LIN {X 0,Y 469.267,Z 468.198,A -85,B 0,C 180,E1 -7456.775,E2 -7456.775} C_VEL
LIN {X 0,Y 468.626,Z 477.541,A -85,B 0,C 180,E1 -7458.1,E2 -7458.1} C_VEL
LIN {X 0,Y 468.005,Z 486.29,A -85,B 0,C 180,E1 -7459.618,E2 -7459.618} C_VEL
LIN {X 0,Y 467.579,Z 492.456,A -85,B 0,C 180,E1 -7460.919,E2 -7460.919} C_VEL
LIN {X 0,Y 467.288,Z 497.539,A -85,B 0,C 180,E1 -7462.22,E2 -7462.22} C_VEL
LIN {X 0,Y 467.051,Z 502.915,A -85,B 0,C 180,E1 -7463.953,E2 -7463.953} C_VEL
LIN {X 0,Y 466.841,Z 506.814,A -85,B 0,C 180,E1 -7465.683,E2 -7465.683} C_VEL
LIN {X 0,Y 466.764,Z 509.357,A -85,B 0,C 180,E1 -7467.411,E2 -7467.411} C_VEL
LIN {X 0,Y 466.622,Z 510.634,A -85,B 0,C 180,E1 -7469.137,E2 -7469.137} C_VEL
LIN {X 0,Y 466.622,Z 510.669,A -85,B 0,C 180,E1 -7470.863,E2 -7470.863} C_VEL
LIN {X 0,Y 466.762,Z 509.467,A -85,B 0,C 180,E1 -7472.589,E2 -7472.589} C_VEL
LIN {X 0,Y 466.825,Z 506.997,A -85,B 0,C 180,E1 -7474.317,E2 -7474.317} C_VEL
LIN {X 0,Y 467.046,Z 503.165,A -85,B 0,C 180,E1 -7476.046,E2 -7476.046} C_VEL
LIN {X 0,Y 467.237,Z 497.87,A -85,B 0,C 180,E1 -7477.78,E2 -7477.78} C_VEL
LIN {X 0,Y 467.649,Z 490.923,A -85,B 0,C 180,E1 -7479.515,E2 -7479.515} C_VEL
LIN {X 0,Y 468.194,Z 483.257,A -85,B 0,C 180,E1 -7481.033,E2 -7481.033} C_VEL
LIN {X 0,Y 468.792,Z 475.255,A -85,B 0,C 180,E1 -7482.335,E2 -7482.335} C_VEL
LIN {X 0,Y 469.426,Z 465.627,A -85,B 0,C 180,E1 -7483.638,E2 -7483.638} C_VEL
LIN {X 0,Y 470.223,Z 454.915,A -85,B 0,C 180,E1 -7484.829,E2 -7484.829} C_VEL
LIN {X 0,Y 471,Z 443.033,A -85,B 0,C 180,E1 -7485.913,E2 -7485.913} C_VEL
LIN {X 0,Y 471.72,Z 431.29,A -85,B 0,C 180,E1 -7486.777,E2 -7486.777} C_VEL
LIN {X 0,Y 472.372,Z 418.989,A -85,B 0,C 180,E1 -7487.5,E2 -7487.5} C_VEL
LIN {X 0,Y 472.878,Z 404.897,A -85,B 0,C 180,E1 -7488.135,E2 -7488.135} C_VEL
LIN {X 0,Y 473.318,Z 391.368,A -85,B 0,C 180,E1 -7488.56,E2 -7488.56} C_VEL
LIN {X 0,Y 473.564,Z 375.614,A -85,B 0,C 180,E1 -7488.859,E2 -7488.859} C_VEL
LIN {X 0,Y 474.304,Z 263.513,A -85,B 0,C 180,E1 -7490.488,E2 -7490.488} C_VEL
LIN {X 0,Y 470.511,Z 244.594,A -85,B 0,C 180,E1 -7490.98,E2 -7490.98} C_VEL
LIN {X 0,Y 470.717,Z 239.725,A -85,B 0,C 180,E1 -7491.686,E2 -7491.686} C_VEL
LIN {X 0,Y 472.048,Z 216.347,A -85,B 0,C 180,E1 -7495.342,E2 -7495.342} C_VEL
LIN {X 0,Y 471.922,Z 212.053,A -85,B 0,C 180,E1 -7496.045,E2 -7496.045} C_VEL
LIN {X 0,Y 468.466,Z 197.446,A -85,B 0,C 180,E1 -7498.689,E2 -7498.689} C_VEL
LIN {X 0,Y 467.573,Z 193.923,A -85,B 0,C 180,E1 -7499.4,E2 -7499.4} C_VEL
LIN {X 0,Y 467.582,Z 193.852,A -85,B 0,C 180,E1 -7502.758,E2 -7502.758} C_VEL
LIN {X 0,Y 467.554,Z 193.869,A -85,B 0,C 180,E1 -7505.889,E2 -7505.889} C_VEL
LIN {X 0,Y 467.58,Z 193.863,A -85,B 0,C 180,E1 -7509.144,E2 -7509.144} C_VEL
LIN {X 0,Y 467.583,Z 193.858,A -85,B 0,C 180,E1 -7512.566,E2 -7512.566} C_VEL
LIN {X 0,Y 467.567,Z 193.867,A -85,B 0,C 180,E1 -7515.052,E2 -7515.052} C_VEL
LIN {X 0,Y 467.585,Z 193.867,A -85,B 0,C 180,E1 -7517.439,E2 -7517.439} C_VEL
LIN {X 0,Y 467.556,Z 193.86,A -85,B 0,C 180,E1 -7520.852,E2 -7520.852} C_VEL
LIN {X 0,Y 467.558,Z 193.862,A -85,B 0,C 180,E1 -7524.26,E2 -7524.26} C_VEL
LIN {X 0,Y 467.577,Z 193.868,A -85,B 0,C 180,E1 -7527.32,E2 -7527.32} C_VEL
LIN {X 0,Y 467.573,Z 193.857,A -85,B 0,C 180,E1 -7530.665,E2 -7530.665} C_VEL
LIN {X 0,Y 467.611,Z 193.86,A -85,B 0,C 180,E1 -7533.199,E2 -7533.199} C_VEL
LIN {X 0,Y 467.586,Z 193.861,A -85,B 0,C 180,E1 -7536.468,E2 -7536.468} C_VEL
LIN {X 0,Y 467.616,Z 193.854,A -85,B 0,C 180,E1 -7539.777,E2 -7539.777} C_VEL
LIN {X 0,Y 467.603,Z 193.864,A -85,B 0,C 180,E1 -7542.506,E2 -7542.506} C_VEL
LIN {X 0,Y 467.601,Z 193.863,A -85,B 0,C 180,E1 -7545.196,E2 -7545.196} C_VEL
LIN {X 0,Y 467.649,Z 193.851,A -85,B 0,C 180,E1 -7547.854,E2 -7547.854} C_VEL
LIN {X 0,Y 467.675,Z 193.849,A -85,B 0,C 180,E1 -7551.357,E2 -7551.357} C_VEL
LIN {X 0,Y 467.736,Z 193.843,A -85,B 0,C 180,E1 -7553.962,E2 -7553.962} C_VEL
LIN {X 0,Y 467.853,Z 193.826,A -85,B 0,C 180,E1 -7557.417,E2 -7557.417} C_VEL
LIN {X 0,Y 467.875,Z 193.829,A -85,B 0,C 180,E1 -7560,E2 -7560} C_VEL
LIN {X 0,Y 467.853,Z 193.834,A -85,B 0,C 180,E1 -7562.583,E2 -7562.583} C_VEL
LIN {X 0,Y 467.736,Z 193.843,A -85,B 0,C 180,E1 -7566.037,E2 -7566.037} C_VEL
LIN {X 0,Y 467.674,Z 193.851,A -85,B 0,C 180,E1 -7568.643,E2 -7568.643} C_VEL
LIN {X 0,Y 467.648,Z 193.86,A -85,B 0,C 180,E1 -7572.145,E2 -7572.145} C_VEL
LIN {X 0,Y 467.631,Z 193.859,A -85,B 0,C 180,E1 -7575.695,E2 -7575.695} C_VEL
LIN {X 0,Y 467.61,Z 193.858,A -85,B 0,C 180,E1 -7578.765,E2 -7578.765} C_VEL
LIN {X 0,Y 467.573,Z 193.863,A -85,B 0,C 180,E1 -7581.268,E2 -7581.268} C_VEL
LIN {X 0,Y 467.566,Z 193.867,A -85,B 0,C 180,E1 -7583.943,E2 -7583.943} C_VEL
LIN {X 0,Y 467.612,Z 193.845,A -85,B 0,C 180,E1 -7586.8,E2 -7586.8} C_VEL
LIN {X 0,Y 467.546,Z 193.873,A -85,B 0,C 180,E1 -7589.739,E2 -7589.739} C_VEL
LIN {X 0,Y 467.577,Z 193.851,A -85,B 0,C 180,E1 -7592.759,E2 -7592.759} C_VEL
LIN {X 0,Y 467.55,Z 193.867,A -85,B 0,C 180,E1 -7595.89,E2 -7595.89} C_VEL
LIN {X 0,Y 467.576,Z 193.864,A -85,B 0,C 180,E1 -7599.145,E2 -7599.145} C_VEL
LIN {X 0,Y 467.581,Z 193.859,A -85,B 0,C 180,E1 -7602.567,E2 -7602.567} C_VEL
LIN {X 0,Y 467.56,Z 193.867,A -85,B 0,C 180,E1 -7605.053,E2 -7605.053} C_VEL
LIN {X 0,Y 467.584,Z 193.867,A -85,B 0,C 180,E1 -7607.441,E2 -7607.441} C_VEL
LIN {X 0,Y 467.554,Z 193.848,A -85,B 0,C 180,E1 -7610.853,E2 -7610.853} C_VEL
LIN {X 0,Y 467.555,Z 193.855,A -85,B 0,C 180,E1 -7614.262,E2 -7614.262} C_VEL
LIN {X 0,Y 467.569,Z 193.861,A -85,B 0,C 180,E1 -7617.323,E2 -7617.323} C_VEL
LIN {X 0,Y 467.574,Z 194.014,A -85,B 0,C 180,E1 -7619.018,E2 -7619.018} C_VEL
LIN {X 0,Y 470.497,Z 204.521,A -85,B 0,C 180,E1 -7620.713,E2 -7620.713} C_VEL
LIN {X 0,Y 473.464,Z 217.047,A -85,B 0,C 180,E1 -7622.604,E2 -7622.604} C_VEL
LIN {X 0,Y 471.777,Z 243.748,A -85,B 0,C 180,E1 -7626.051,E2 -7626.051} C_VEL
LIN {X 0,Y 471.739,Z 245.311,A -85,B 0,C 180,E1 -7626.211,E2 -7626.211} C_VEL
LIN {X 0,Y 475.092,Z 265.679,A -85,B 0,C 180,E1 -7626.729,E2 -7626.729} C_VEL
LIN {X 0,Y 473.209,Z 408.687,A -85,B 0,C 180,E1 -7629.062,E2 -7629.062} C_VEL
LIN {X 0,Y 472.673,Z 424.604,A -85,B 0,C 180,E1 -7629.491,E2 -7629.491} C_VEL
LIN {X 0,Y 472.053,Z 439.866,A -85,B 0,C 180,E1 -7630.089,E2 -7630.089} C_VEL
LIN {X 0,Y 471.299,Z 454.544,A -85,B 0,C 180,E1 -7630.849,E2 -7630.849} C_VEL
LIN {X 0,Y 470.534,Z 467.938,A -85,B 0,C 180,E1 -7631.721,E2 -7631.721} C_VEL
LIN {X 0,Y 469.794,Z 481.582,A -85,B 0,C 180,E1 -7632.816,E2 -7632.816} C_VEL
LIN {X 0,Y 469.075,Z 493.997,A -85,B 0,C 180,E1 -7634.02,E2 -7634.02} C_VEL
LIN {X 0,Y 468.418,Z 504.464,A -85,B 0,C 180,E1 -7635.223,E2 -7635.223} C_VEL
LIN {X 0,Y 467.834,Z 515.629,A -85,B 0,C 180,E1 -7636.757,E2 -7636.757} C_VEL
LIN {X 0,Y 467.425,Z 524.894,A -85,B 0,C 180,E1 -7638.289,E2 -7638.289} C_VEL
LIN {X 0,Y 467.087,Z 532.575,A -85,B 0,C 180,E1 -7639.817,E2 -7639.817} C_VEL
LIN {X 0,Y 466.875,Z 538.894,A -85,B 0,C 180,E1 -7641.343,E2 -7641.343} C_VEL
LIN {X 0,Y 466.758,Z 544.686,A -85,B 0,C 180,E1 -7643.082,E2 -7643.082} C_VEL
LIN {X 0,Y 466.717,Z 549.068,A -85,B 0,C 180,E1 -7644.817,E2 -7644.817} C_VEL
LIN {X 0,Y 466.706,Z 552.142,A -85,B 0,C 180,E1 -7646.547,E2 -7646.547} C_VEL
LIN {X 0,Y 466.658,Z 553.973,A -85,B 0,C 180,E1 -7648.274,E2 -7648.274} C_VEL
LIN {X 0,Y 466.597,Z 554.595,A -85,B 0,C 180,E1 -7650,E2 -7650} C_VEL
LIN {X 0,Y 466.658,Z 553.97,A -85,B 0,C 180,E1 -7651.726,E2 -7651.726} C_VEL
LIN {X 0,Y 466.706,Z 552.136,A -85,B 0,C 180,E1 -7653.454,E2 -7653.454} C_VEL
LIN {X 0,Y 466.722,Z 549.065,A -85,B 0,C 180,E1 -7655.184,E2 -7655.184} C_VEL
LIN {X 0,Y 466.821,Z 544.69,A -85,B 0,C 180,E1 -7656.918,E2 -7656.918} C_VEL
LIN {X 0,Y 466.875,Z 538.89,A -85,B 0,C 180,E1 -7658.658,E2 -7658.658} C_VEL
LIN {X 0,Y 467.179,Z 531.526,A -85,B 0,C 180,E1 -7660.4,E2 -7660.4} C_VEL
LIN {X 0,Y 467.477,Z 523.63,A -85,B 0,C 180,E1 -7661.93,E2 -7661.93} C_VEL
LIN {X 0,Y 467.919,Z 514.123,A -85,B 0,C 180,E1 -7663.462,E2 -7663.462} C_VEL
LIN {X 0,Y 468.413,Z 504.449,A -85,B 0,C 180,E1 -7664.778,E2 -7664.778} C_VEL
LIN {X 0,Y 469.096,Z 492.954,A -85,B 0,C 180,E1 -7666.091,E2 -7666.091} C_VEL
LIN {X 0,Y 469.869,Z 480.323,A -85,B 0,C 180,E1 -7667.294,E2 -7667.294} C_VEL
LIN {X 0,Y 470.543,Z 467.908,A -85,B 0,C 180,E1 -7668.28,E2 -7668.28} C_VEL
LIN {X 0,Y 471.313,Z 454.501,A -85,B 0,C 180,E1 -7669.151,E2 -7669.151} C_VEL
LIN {X 0,Y 472.067,Z 439.828,A -85,B 0,C 180,E1 -7669.911,E2 -7669.911} C_VEL
LIN {X 0,Y 472.701,Z 424.193,A -85,B 0,C 180,E1 -7670.521,E2 -7670.521} C_VEL
LIN {X 0,Y 473.161,Z 408.552,A -85,B 0,C 180,E1 -7670.941,E2 -7670.941} C_VEL
LIN {X 0,Y 475.017,Z 270.123,A -85,B 0,C 180,E1 -7673.198,E2 -7673.198} C_VEL
LIN {X 0,Y 474.917,Z 264.066,A -85,B 0,C 180,E1 -7673.304,E2 -7673.304} C_VEL
LIN {X 0,Y 471.704,Z 245.037,A -85,B 0,C 180,E1 -7673.801,E2 -7673.801} C_VEL
LIN {X 0,Y 473.005,Z 224.215,A -85,B 0,C 180,E1 -7676.471,E2 -7676.471} C_VEL
LIN {X 0,Y 473.439,Z 217.06,A -85,B 0,C 180,E1 -7677.399,E2 -7677.399} C_VEL
LIN {X 0,Y 470.952,Z 206.283,A -85,B 0,C 180,E1 -7679.012,E2 -7679.012} C_VEL
LIN {X 0,Y 467.576,Z 193.975,A -85,B 0,C 180,E1 -7680.983,E2 -7680.983} C_VEL
LIN {X 0,Y 467.575,Z 193.857,A -85,B 0,C 180,E1 -7684.24,E2 -7684.24} C_VEL
LIN {X 0,Y 467.546,Z 193.873,A -85,B 0,C 180,E1 -7687.186,E2 -7687.186} C_VEL
LIN {X 0,Y 467.572,Z 193.842,A -85,B 0,C 180,E1 -7690.265,E2 -7690.265} C_VEL
LIN {X 0,Y 467.585,Z 193.867,A -85,B 0,C 180,E1 -7692.567,E2 -7692.567} C_VEL
LIN {X 0,Y 467.564,Z 193.867,A -85,B 0,C 180,E1 -7695.052,E2 -7695.052} C_VEL
LIN {X 0,Y 467.587,Z 193.858,A -85,B 0,C 180,E1 -7697.44,E2 -7697.44} C_VEL
LIN {X 0,Y 467.58,Z 193.864,A -85,B 0,C 180,E1 -7700.855,E2 -7700.855} C_VEL
LIN {X 0,Y 467.557,Z 193.869,A -85,B 0,C 180,E1 -7704.261,E2 -7704.261} C_VEL
LIN {X 0,Y 467.579,Z 193.851,A -85,B 0,C 180,E1 -7707.321,E2 -7707.321} C_VEL
LIN {X 0,Y 467.566,Z 193.867,A -85,B 0,C 180,E1 -7710.668,E2 -7710.668} C_VEL
LIN {X 0,Y 467.61,Z 193.844,A -85,B 0,C 180,E1 -7713.199,E2 -7713.199} C_VEL
LIN {X 0,Y 467.588,Z 193.866,A -85,B 0,C 180,E1 -7716.469,E2 -7716.469} C_VEL
LIN {X 0,Y 467.62,Z 193.859,A -85,B 0,C 180,E1 -7719.777,E2 -7719.777} C_VEL
LIN {X 0,Y 467.605,Z 193.861,A -85,B 0,C 180,E1 -7722.507,E2 -7722.507} C_VEL
LIN {X 0,Y 467.603,Z 193.859,A -85,B 0,C 180,E1 -7725.197,E2 -7725.197} C_VEL
LIN {X 0,Y 467.653,Z 193.859,A -85,B 0,C 180,E1 -7727.855,E2 -7727.855} C_VEL
LIN {X 0,Y 467.678,Z 193.85,A -85,B 0,C 180,E1 -7731.357,E2 -7731.357} C_VEL
LIN {X 0,Y 467.74,Z 193.843,A -85,B 0,C 180,E1 -7733.963,E2 -7733.963} C_VEL
LIN {X 0,Y 467.856,Z 193.833,A -85,B 0,C 180,E1 -7737.417,E2 -7737.417} C_VEL
LIN {X 0,Y 467.879,Z 193.829,A -85,B 0,C 180,E1 -7740,E2 -7740} C_VEL
LIN {X 0,Y 467.857,Z 193.825,A -85,B 0,C 180,E1 -7742.583,E2 -7742.583} C_VEL
LIN {X 0,Y 467.741,Z 193.843,A -85,B 0,C 180,E1 -7746.038,E2 -7746.038} C_VEL
LIN {X 0,Y 467.679,Z 193.849,A -85,B 0,C 180,E1 -7748.643,E2 -7748.643} C_VEL
LIN {X 0,Y 467.653,Z 193.85,A -85,B 0,C 180,E1 -7752.146,E2 -7752.146} C_VEL
LIN {X 0,Y 467.637,Z 193.854,A -85,B 0,C 180,E1 -7755.695,E2 -7755.695} C_VEL
LIN {X 0,Y 467.615,Z 193.861,A -85,B 0,C 180,E1 -7758.765,E2 -7758.765} C_VEL
LIN {X 0,Y 467.578,Z 193.869,A -85,B 0,C 180,E1 -7761.268,E2 -7761.268} C_VEL
LIN {X 0,Y 467.57,Z 193.862,A -85,B 0,C 180,E1 -7763.944,E2 -7763.944} C_VEL
LIN {X 0,Y 467.615,Z 193.861,A -85,B 0,C 180,E1 -7766.801,E2 -7766.801} C_VEL
LIN {X 0,Y 467.552,Z 193.86,A -85,B 0,C 180,E1 -7769.738,E2 -7769.738} C_VEL
LIN {X 0,Y 467.582,Z 193.867,A -85,B 0,C 180,E1 -7772.759,E2 -7772.759} C_VEL
LIN {X 0,Y 467.556,Z 193.861,A -85,B 0,C 180,E1 -7775.89,E2 -7775.89} C_VEL
LIN {X 0,Y 467.559,Z 193.859,A -85,B 0,C 180,E1 -7779.147,E2 -7779.147} C_VEL
LIN {X 0,Y 467.586,Z 193.868,A -85,B 0,C 180,E1 -7782.567,E2 -7782.567} C_VEL
LIN {X 0,Y 467.571,Z 193.867,A -85,B 0,C 180,E1 -7785.053,E2 -7785.053} C_VEL
LIN {X 0,Y 467.589,Z 193.858,A -85,B 0,C 180,E1 -7787.44,E2 -7787.44} C_VEL
LIN {X 0,Y 467.582,Z 193.862,A -85,B 0,C 180,E1 -7790.856,E2 -7790.856} C_VEL
LIN {X 0,Y 467.562,Z 193.869,A -85,B 0,C 180,E1 -7794.261,E2 -7794.261} C_VEL
LIN {X 0,Y 467.583,Z 193.851,A -85,B 0,C 180,E1 -7797.321,E2 -7797.321} C_VEL
LIN {X 0,Y 467.586,Z 193.972,A -85,B 0,C 180,E1 -7800.732,E2 -7800.732} C_VEL
LIN {X 0,Y 470.786,Z 207.019,A -85,B 0,C 180,E1 -7803.155,E2 -7803.155} C_VEL
LIN {X 0,Y 472.11,Z 212.897,A -85,B 0,C 180,E1 -7804.201,E2 -7804.201} C_VEL
LIN {X 0,Y 471.337,Z 227.381,A -85,B 0,C 180,E1 -7806.493,E2 -7806.493} C_VEL
LIN {X 0,Y 470.478,Z 244.431,A -85,B 0,C 180,E1 -7809.102,E2 -7809.102} C_VEL
LIN {X 0,Y 474.392,Z 264.64,A -85,B 0,C 180,E1 -7809.626,E2 -7809.626} C_VEL
LIN {X 0,Y 474.417,Z 267.518,A -85,B 0,C 180,E1 -7809.67,E2 -7809.67} C_VEL
LIN {X 0,Y 473.774,Z 273.373,A -85,B 0,C 180,E1 -7809.728,E2 -7809.728} C_VEL
LIN {X 0,Y 468.182,Z 292.425,A -85,B 0,C 180,E1 -7809.744,E2 -7809.744} C_VEL
LIN {X 0,Y 467.551,Z 298.281,A -85,B 0,C 180,E1 -7809.802,E2 -7809.802} C_VEL
LIN {X 0,Y 466.805,Z 384.962,A -85,B 0,C 180,E1 -7811.085,E2 -7811.085} C_VEL
LIN {X 0,Y 466.403,Z 399.475,A -85,B 0,C 180,E1 -7811.467,E2 -7811.467} C_VEL
LIN {X 0,Y 465.951,Z 413.371,A -85,B 0,C 180,E1 -7812.023,E2 -7812.023} C_VEL
LIN {X 0,Y 465.404,Z 425.207,A -85,B 0,C 180,E1 -7812.648,E2 -7812.648} C_VEL
LIN {X 0,Y 464.569,Z 438.207,A -85,B 0,C 180,E1 -7813.522,E2 -7813.522} C_VEL
LIN {X 0,Y 463.756,Z 449.946,A -85,B 0,C 180,E1 -7814.508,E2 -7814.508} C_VEL
LIN {X 0,Y 463.052,Z 459.693,A -85,B 0,C 180,E1 -7815.497,E2 -7815.497} C_VEL
LIN {X 0,Y 462.234,Z 470.42,A -85,B 0,C 180,E1 -7816.817,E2 -7816.817} C_VEL
LIN {X 0,Y 461.554,Z 479.282,A -85,B 0,C 180,E1 -7818.137,E2 -7818.137} C_VEL
LIN {X 0,Y 460.921,Z 487.753,A -85,B 0,C 180,E1 -7819.679,E2 -7819.679} C_VEL
LIN {X 0,Y 460.444,Z 494.611,A -85,B 0,C 180,E1 -7821.22,E2 -7821.22} C_VEL
LIN {X 0,Y 460.07,Z 500.781,A -85,B 0,C 180,E1 -7822.98,E2 -7822.98} C_VEL
LIN {X 0,Y 459.882,Z 504.367,A -85,B 0,C 180,E1 -7824.299,E2 -7824.299} C_VEL
LIN {X 0,Y 459.752,Z 507.157,A -85,B 0,C 180,E1 -7825.616,E2 -7825.616} C_VEL
LIN {X 0,Y 459.683,Z 509.694,A -85,B 0,C 180,E1 -7827.371,E2 -7827.371} C_VEL
LIN {X 0,Y 459.556,Z 510.966,A -85,B 0,C 180,E1 -7829.123,E2 -7829.123} C_VEL
LIN {X 0,Y 459.556,Z 511.001,A -85,B 0,C 180,E1 -7830.876,E2 -7830.876} C_VEL
LIN {X 0,Y 459.68,Z 509.802,A -85,B 0,C 180,E1 -7832.629,E2 -7832.629} C_VEL
LIN {X 0,Y 459.736,Z 507.339,A -85,B 0,C 180,E1 -7834.383,E2 -7834.383} C_VEL
LIN {X 0,Y 460.001,Z 503.513,A -85,B 0,C 180,E1 -7836.139,E2 -7836.139} C_VEL
LIN {X 0,Y 460.209,Z 498.228,A -85,B 0,C 180,E1 -7837.899,E2 -7837.899} C_VEL
LIN {X 0,Y 460.535,Z 493.23,A -85,B 0,C 180,E1 -7839.22,E2 -7839.22} C_VEL
LIN {X 0,Y 461.08,Z 486.029,A -85,B 0,C 180,E1 -7840.761,E2 -7840.761} C_VEL
LIN {X 0,Y 461.627,Z 478.513,A -85,B 0,C 180,E1 -7842.083,E2 -7842.083} C_VEL
LIN {X 0,Y 462.328,Z 468.945,A -85,B 0,C 180,E1 -7843.479,E2 -7843.479} C_VEL
LIN {X 0,Y 463.096,Z 458.514,A -85,B 0,C 180,E1 -7844.726,E2 -7844.726} C_VEL
LIN {X 0,Y 463.91,Z 447.333,A -85,B 0,C 180,E1 -7845.824,E2 -7845.824} C_VEL
LIN {X 0,Y 464.779,Z 434.949,A -85,B 0,C 180,E1 -7846.809,E2 -7846.809} C_VEL
LIN {X 0,Y 465.402,Z 422.958,A -85,B 0,C 180,E1 -7847.578,E2 -7847.578} C_VEL
LIN {X 0,Y 466.095,Z 409.337,A -85,B 0,C 180,E1 -7848.248,E2 -7848.248} C_VEL
LIN {X 0,Y 466.529,Z 395.19,A -85,B 0,C 180,E1 -7848.755,E2 -7848.755} C_VEL
LIN {X 0,Y 466.852,Z 380.668,A -85,B 0,C 180,E1 -7849.083,E2 -7849.083} C_VEL
LIN {X 0,Y 467.834,Z 265.856,A -85,B 0,C 180,E1 -7850.771,E2 -7850.771} C_VEL
LIN {X 0,Y 463.8,Z 245.038,A -85,B 0,C 180,E1 -7851.306,E2 -7851.306} C_VEL
LIN {X 0,Y 463.686,Z 243.548,A -85,B 0,C 180,E1 -7851.447,E2 -7851.447} C_VEL
LIN {X 0,Y 464.914,Z 222.567,A -85,B 0,C 180,E1 -7854.762,E2 -7854.762} C_VEL
LIN {X 0,Y 465.323,Z 215.002,A -85,B 0,C 180,E1 -7855.976,E2 -7855.976} C_VEL
LIN {X 0,Y 461.978,Z 200.465,A -85,B 0,C 180,E1 -7858.632,E2 -7858.632} C_VEL
LIN {X 0,Y 460.532,Z 194.804,A -85,B 0,C 180,E1 -7859.758,E2 -7859.758} C_VEL
LIN {X 0,Y 460.529,Z 194.728,A -85,B 0,C 180,E1 -7862.929,E2 -7862.929} C_VEL
LIN {X 0,Y 460.498,Z 194.746,A -85,B 0,C 180,E1 -7866.014,E2 -7866.014} C_VEL
LIN {X 0,Y 460.542,Z 194.74,A -85,B 0,C 180,E1 -7868.897,E2 -7868.897} C_VEL
LIN {X 0,Y 460.52,Z 194.739,A -85,B 0,C 180,E1 -7872.181,E2 -7872.181} C_VEL
LIN {X 0,Y 460.513,Z 194.742,A -85,B 0,C 180,E1 -7875.411,E2 -7875.411} C_VEL
LIN {X 0,Y 460.528,Z 194.743,A -85,B 0,C 180,E1 -7878.397,E2 -7878.397} C_VEL
LIN {X 0,Y 460.514,Z 194.741,A -85,B 0,C 180,E1 -7881.266,E2 -7881.266} C_VEL
LIN {X 0,Y 460.509,Z 194.741,A -85,B 0,C 180,E1 -7884.554,E2 -7884.554} C_VEL
LIN {X 0,Y 460.527,Z 194.744,A -85,B 0,C 180,E1 -7887.715,E2 -7887.715} C_VEL
LIN {X 0,Y 460.542,Z 194.731,A -85,B 0,C 180,E1 -7890.769,E2 -7890.769} C_VEL
LIN {X 0,Y 460.557,Z 194.738,A -85,B 0,C 180,E1 -7893.734,E2 -7893.734} C_VEL
LIN {X 0,Y 460.54,Z 194.74,A -85,B 0,C 180,E1 -7896.623,E2 -7896.623} C_VEL
LIN {X 0,Y 460.544,Z 194.737,A -85,B 0,C 180,E1 -7899.452,E2 -7899.452} C_VEL
LIN {X 0,Y 460.553,Z 194.739,A -85,B 0,C 180,E1 -7902.23,E2 -7902.23} C_VEL
LIN {X 0,Y 460.559,Z 194.742,A -85,B 0,C 180,E1 -7904.964,E2 -7904.964} C_VEL
LIN {X 0,Y 460.602,Z 194.729,A -85,B 0,C 180,E1 -7907.665,E2 -7907.665} C_VEL
LIN {X 0,Y 460.622,Z 194.729,A -85,B 0,C 180,E1 -7911.224,E2 -7911.224} C_VEL
LIN {X 0,Y 460.703,Z 194.719,A -85,B 0,C 180,E1 -7913.87,E2 -7913.87} C_VEL
LIN {X 0,Y 460.818,Z 194.702,A -85,B 0,C 180,E1 -7917.377,E2 -7917.377} C_VEL
LIN {X 0,Y 460.845,Z 194.704,A -85,B 0,C 180,E1 -7920,E2 -7920} C_VEL
LIN {X 0,Y 460.818,Z 194.71,A -85,B 0,C 180,E1 -7922.622,E2 -7922.622} C_VEL
LIN {X 0,Y 460.703,Z 194.719,A -85,B 0,C 180,E1 -7926.13,E2 -7926.13} C_VEL
LIN {X 0,Y 460.621,Z 194.728,A -85,B 0,C 180,E1 -7928.776,E2 -7928.776} C_VEL
LIN {X 0,Y 460.606,Z 194.733,A -85,B 0,C 180,E1 -7932.445,E2 -7932.445} C_VEL
LIN {X 0,Y 460.592,Z 194.74,A -85,B 0,C 180,E1 -7935.998,E2 -7935.998} C_VEL
LIN {X 0,Y 460.563,Z 194.736,A -85,B 0,C 180,E1 -7938.902,E2 -7938.902} C_VEL
LIN {X 0,Y 460.508,Z 194.744,A -85,B 0,C 180,E1 -7941.486,E2 -7941.486} C_VEL
LIN {X 0,Y 460.536,Z 194.739,A -85,B 0,C 180,E1 -7944.332,E2 -7944.332} C_VEL
LIN {X 0,Y 460.573,Z 194.723,A -85,B 0,C 180,E1 -7947.244,E2 -7947.244} C_VEL
LIN {X 0,Y 460.503,Z 194.745,A -85,B 0,C 180,E1 -7950.24,E2 -7950.24} C_VEL
LIN {X 0,Y 460.523,Z 194.734,A -85,B 0,C 180,E1 -7953.325,E2 -7953.325} C_VEL
LIN {X 0,Y 460.472,Z 194.746,A -85,B 0,C 180,E1 -7956.53,E2 -7956.53} C_VEL
LIN {X 0,Y 460.552,Z 194.742,A -85,B 0,C 180,E1 -7959.86,E2 -7959.86} C_VEL
LIN {X 0,Y 460.506,Z 194.742,A -85,B 0,C 180,E1 -7962.901,E2 -7962.901} C_VEL
LIN {X 0,Y 460.503,Z 194.743,A -85,B 0,C 180,E1 -7965.831,E2 -7965.831} C_VEL
LIN {X 0,Y 460.525,Z 194.728,A -85,B 0,C 180,E1 -7968.989,E2 -7968.989} C_VEL
LIN {X 0,Y 460.513,Z 194.73,A -85,B 0,C 180,E1 -7971.267,E2 -7971.267} C_VEL
LIN {X 0,Y 460.504,Z 194.73,A -85,B 0,C 180,E1 -7974.555,E2 -7974.555} C_VEL
LIN {X 0,Y 460.514,Z 194.719,A -85,B 0,C 180,E1 -7977.715,E2 -7977.715} C_VEL
LIN {X 0,Y 460.577,Z 194.958,A -85,B 0,C 180,E1 -7978.662,E2 -7978.662} C_VEL
LIN {X 0,Y 464.137,Z 208.021,A -85,B 0,C 180,E1 -7980.777,E2 -7980.777} C_VEL
LIN {X 0,Y 466.622,Z 218.341,A -85,B 0,C 180,E1 -7982.366,E2 -7982.366} C_VEL
LIN {X 0,Y 465.289,Z 240.561,A -85,B 0,C 180,E1 -7985.294,E2 -7985.294} C_VEL
LIN {X 0,Y 464.98,Z 245.065,A -85,B 0,C 180,E1 -7985.857,E2 -7985.857} C_VEL
LIN {X 0,Y 468.54,Z 267.054,A -85,B 0,C 180,E1 -7986.431,E2 -7986.431} C_VEL
LIN {X 0,Y 466.521,Z 408.803,A -85,B 0,C 180,E1 -7988.776,E2 -7988.776} C_VEL
LIN {X 0,Y 465.944,Z 424.716,A -85,B 0,C 180,E1 -7989.215,E2 -7989.215} C_VEL
LIN {X 0,Y 465.359,Z 439.202,A -85,B 0,C 180,E1 -7989.79,E2 -7989.79} C_VEL
LIN {X 0,Y 464.533,Z 453.968,A -85,B 0,C 180,E1 -7990.559,E2 -7990.559} C_VEL
LIN {X 0,Y 463.725,Z 467.409,A -85,B 0,C 180,E1 -7991.443,E2 -7991.443} C_VEL
LIN {X 0,Y 462.909,Z 481.098,A -85,B 0,C 180,E1 -7992.552,E2 -7992.552} C_VEL
LIN {X 0,Y 462.183,Z 492.772,A -85,B 0,C 180,E1 -7993.69,E2 -7993.69} C_VEL
LIN {X 0,Y 461.456,Z 504.023,A -85,B 0,C 180,E1 -7994.995,E2 -7994.995} C_VEL
LIN {X 0,Y 460.832,Z 515.218,A -85,B 0,C 180,E1 -7996.552,E2 -7996.552} C_VEL
LIN {X 0,Y 460.351,Z 524.661,A -85,B 0,C 180,E1 -7998.137,E2 -7998.137} C_VEL
LIN {X 0,Y 460.06,Z 532.193,A -85,B 0,C 180,E1 -7999.66,E2 -7999.66} C_VEL
LIN {X 0,Y 459.81,Z 538.525,A -85,B 0,C 180,E1 -8001.209,E2 -8001.209} C_VEL
LIN {X 0,Y 459.69,Z 544.329,A -85,B 0,C 180,E1 -8002.975,E2 -8002.975} C_VEL
LIN {X 0,Y 459.622,Z 548.721,A -85,B 0,C 180,E1 -8004.736,E2 -8004.736} C_VEL
LIN {X 0,Y 459.601,Z 551.802,A -85,B 0,C 180,E1 -8006.494,E2 -8006.494} C_VEL
LIN {X 0,Y 459.567,Z 553.639,A -85,B 0,C 180,E1 -8008.248,E2 -8008.248} C_VEL
LIN {X 0,Y 459.528,Z 554.263,A -85,B 0,C 180,E1 -8010,E2 -8010} C_VEL
LIN {X 0,Y 459.567,Z 553.636,A -85,B 0,C 180,E1 -8011.753,E2 -8011.753} C_VEL
LIN {X 0,Y 459.601,Z 551.796,A -85,B 0,C 180,E1 -8013.507,E2 -8013.507} C_VEL
LIN {X 0,Y 459.633,Z 548.717,A -85,B 0,C 180,E1 -8015.264,E2 -8015.264} C_VEL
LIN {X 0,Y 459.728,Z 544.331,A -85,B 0,C 180,E1 -8017.025,E2 -8017.025} C_VEL
LIN {X 0,Y 459.811,Z 538.519,A -85,B 0,C 180,E1 -8018.792,E2 -8018.792} C_VEL
LIN {X 0,Y 460.102,Z 531.138,A -85,B 0,C 180,E1 -8020.562,E2 -8020.562} C_VEL
LIN {X 0,Y 460.446,Z 522.769,A -85,B 0,C 180,E1 -8022.196,E2 -8022.196} C_VEL
LIN {X 0,Y 460.935,Z 513.702,A -85,B 0,C 180,E1 -8023.67,E2 -8023.67} C_VEL
LIN {X 0,Y 461.447,Z 504.004,A -85,B 0,C 180,E1 -8025.006,E2 -8025.006} C_VEL
LIN {X 0,Y 462.118,Z 492.743,A -85,B 0,C 180,E1 -8026.313,E2 -8026.313} C_VEL
LIN {X 0,Y 463.007,Z 479.814,A -85,B 0,C 180,E1 -8027.559,E2 -8027.559} C_VEL
LIN {X 0,Y 463.744,Z 467.371,A -85,B 0,C 180,E1 -8028.557,E2 -8028.557} C_VEL
LIN {X 0,Y 464.544,Z 453.916,A -85,B 0,C 180,E1 -8029.441,E2 -8029.441} C_VEL
LIN {X 0,Y 465.309,Z 439.145,A -85,B 0,C 180,E1 -8030.213,E2 -8030.213} C_VEL
LIN {X 0,Y 466.003,Z 423.834,A -85,B 0,C 180,E1 -8030.812,E2 -8030.812} C_VEL
LIN {X 0,Y 466.473,Z 408.654,A -85,B 0,C 180,E1 -8031.227,E2 -8031.227} C_VEL
LIN {X 0,Y 468.214,Z 286.116,A -85,B 0,C 180,E1 -8033.258,E2 -8033.258} C_VEL
LIN {X 0,Y 468.341,Z 265.157,A -85,B 0,C 180,E1 -8033.608,E2 -8033.608} C_VEL
LIN {X 0,Y 464.97,Z 245.006,A -85,B 0,C 180,E1 -8034.145,E2 -8034.145} C_VEL
LIN {X 0,Y 466.625,Z 220.822,A -85,B 0,C 180,E1 -8037.3,E2 -8037.3} C_VEL
LIN {X 0,Y 466.355,Z 216.897,A -85,B 0,C 180,E1 -8037.851,E2 -8037.851} C_VEL
LIN {X 0,Y 462.711,Z 202.567,A -85,B 0,C 180,E1 -8040.081,E2 -8040.081} C_VEL
LIN {X 0,Y 460.536,Z 194.836,A -85,B 0,C 180,E1 -8041.37,E2 -8041.37} C_VEL
LIN {X 0,Y 460.521,Z 194.731,A -85,B 0,C 180,E1 -8044.504,E2 -8044.504} C_VEL
LIN {X 0,Y 460.499,Z 194.747,A -85,B 0,C 180,E1 -8047.623,E2 -8047.623} C_VEL
LIN {X 0,Y 460.537,Z 194.717,A -85,B 0,C 180,E1 -8050.269,E2 -8050.269} C_VEL
LIN {X 0,Y 460.497,Z 194.746,A -85,B 0,C 180,E1 -8053.375,E2 -8053.375} C_VEL
LIN {X 0,Y 460.495,Z 194.75,A -85,B 0,C 180,E1 -8056.624,E2 -8056.624} C_VEL
LIN {X 0,Y 460.54,Z 194.741,A -85,B 0,C 180,E1 -8059.731,E2 -8059.731} C_VEL
LIN {X 0,Y 460.497,Z 194.741,A -85,B 0,C 180,E1 -8062.524,E2 -8062.524} C_VEL
LIN {X 0,Y 460.544,Z 194.741,A -85,B 0,C 180,E1 -8065.624,E2 -8065.624} C_VEL
LIN {X 0,Y 460.535,Z 194.741,A -85,B 0,C 180,E1 -8068.744,E2 -8068.744} C_VEL
LIN {X 0,Y 460.578,Z 194.729,A -85,B 0,C 180,E1 -8072.254,E2 -8072.254} C_VEL
LIN {X 0,Y 460.536,Z 194.739,A -85,B 0,C 180,E1 -8074.704,E2 -8074.704} C_VEL
LIN {X 0,Y 460.507,Z 194.745,A -85,B 0,C 180,E1 -8077.571,E2 -8077.571} C_VEL
LIN {X 0,Y 460.566,Z 194.74,A -85,B 0,C 180,E1 -8080.385,E2 -8080.385} C_VEL
LIN {X 0,Y 460.562,Z 194.736,A -85,B 0,C 180,E1 -8083.146,E2 -8083.146} C_VEL
LIN {X 0,Y 460.552,Z 194.74,A -85,B 0,C 180,E1 -8085.868,E2 -8085.868} C_VEL
LIN {X 0,Y 460.608,Z 194.732,A -85,B 0,C 180,E1 -8088.559,E2 -8088.559} C_VEL
LIN {X 0,Y 460.692,Z 194.725,A -85,B 0,C 180,E1 -8092.109,E2 -8092.109} C_VEL
LIN {X 0,Y 460.694,Z 194.716,A -85,B 0,C 180,E1 -8094.748,E2 -8094.748} C_VEL
LIN {X 0,Y 460.797,Z 194.712,A -85,B 0,C 180,E1 -8097.378,E2 -8097.378} C_VEL
LIN {X 0,Y 460.849,Z 194.704,A -85,B 0,C 180,E1 -8100,E2 -8100} C_VEL
LIN {X 0,Y 460.798,Z 194.705,A -85,B 0,C 180,E1 -8102.623,E2 -8102.623} C_VEL
LIN {X 0,Y 460.707,Z 194.719,A -85,B 0,C 180,E1 -8106.13,E2 -8106.13} C_VEL
LIN {X 0,Y 460.626,Z 194.728,A -85,B 0,C 180,E1 -8108.776,E2 -8108.776} C_VEL
LIN {X 0,Y 460.611,Z 194.727,A -85,B 0,C 180,E1 -8112.445,E2 -8112.445} C_VEL
LIN {X 0,Y 460.598,Z 194.729,A -85,B 0,C 180,E1 -8115.998,E2 -8115.998} C_VEL
LIN {X 0,Y 460.569,Z 194.741,A -85,B 0,C 180,E1 -8118.902,E2 -8118.902} C_VEL
LIN {X 0,Y 460.514,Z 194.747,A -85,B 0,C 180,E1 -8121.486,E2 -8121.486} C_VEL
LIN {X 0,Y 460.54,Z 194.738,A -85,B 0,C 180,E1 -8124.333,E2 -8124.333} C_VEL
LIN {X 0,Y 460.571,Z 194.731,A -85,B 0,C 180,E1 -8127.244,E2 -8127.244} C_VEL
LIN {X 0,Y 460.509,Z 194.738,A -85,B 0,C 180,E1 -8130.24,E2 -8130.24} C_VEL
LIN {X 0,Y 460.528,Z 194.738,A -85,B 0,C 180,E1 -8133.325,E2 -8133.325} C_VEL
LIN {X 0,Y 460.478,Z 194.748,A -85,B 0,C 180,E1 -8136.529,E2 -8136.529} C_VEL
LIN {X 0,Y 460.534,Z 194.737,A -85,B 0,C 180,E1 -8138.896,E2 -8138.896} C_VEL
LIN {X 0,Y 460.523,Z 194.746,A -85,B 0,C 180,E1 -8142.182,E2 -8142.182} C_VEL
LIN {X 0,Y 460.517,Z 194.743,A -85,B 0,C 180,E1 -8145.412,E2 -8145.412} C_VEL
LIN {X 0,Y 460.532,Z 194.74,A -85,B 0,C 180,E1 -8148.398,E2 -8148.398} C_VEL
LIN {X 0,Y 460.527,Z 194.741,A -85,B 0,C 180,E1 -8151.267,E2 -8151.267} C_VEL
LIN {X 0,Y 460.513,Z 194.75,A -85,B 0,C 180,E1 -8154.555,E2 -8154.555} C_VEL
LIN {X 0,Y 460.533,Z 194.734,A -85,B 0,C 180,E1 -8157.716,E2 -8157.716} C_VEL
LIN {X 0,Y 460.541,Z 194.881,A -85,B 0,C 180,E1 -8160.385,E2 -8160.385} C_VEL
LIN {X 0,Y 463.927,Z 208.594,A -85,B 0,C 180,E1 -8162.969,E2 -8162.969} C_VEL
LIN {X 0,Y 465.359,Z 215.848,A -85,B 0,C 180,E1 -8164.266,E2 -8164.266} C_VEL
LIN {X 0,Y 464.078,Z 236.132,A -85,B 0,C 180,E1 -8167.486,E2 -8167.486} C_VEL
LIN {X 0,Y 463.695,Z 244.608,A -85,B 0,C 180,E1 -8168.768,E2 -8168.768} C_VEL
LIN {X 0,Y 467.809,Z 265.288,A -85,B 0,C 180,E1 -8169.311,E2 -8169.311} C_VEL
LIN {X 0,Y 467.551,Z 298.281,A -85,B 0,C 180,E1 -8169.802,E2 -8169.802} C_VEL
LIN {X 0,Y 466.931,Z 304.132,A -85,B 0,C 180,E1 -8169.86,E2 -8169.86} C_VEL
LIN {X 0,Y 461.408,Z 323.187,A -85,B 0,C 180,E1 -8169.878,E2 -8169.878} C_VEL
LIN {X 0,Y 460.758,Z 329.041,A -85,B 0,C 180,E1 -8169.936,E2 -8169.936} C_VEL
LIN {X 0,Y 460.132,Z 386.161,A -85,B 0,C 180,E1 -8170.8,E2 -8170.8} C_VEL
LIN {X 0,Y 459.741,Z 400.269,A -85,B 0,C 180,E1 -8171.188,E2 -8171.188} C_VEL
LIN {X 0,Y 459.24,Z 414.275,A -85,B 0,C 180,E1 -8171.764,E2 -8171.764} C_VEL
LIN {X 0,Y 458.711,Z 423.895,A -85,B 0,C 180,E1 -8172.271,E2 -8172.271} C_VEL
LIN {X 0,Y 457.92,Z 437.292,A -85,B 0,C 180,E1 -8173.161,E2 -8173.161} C_VEL
LIN {X 0,Y 457.035,Z 449.254,A -85,B 0,C 180,E1 -8174.16,E2 -8174.16} C_VEL
LIN {X 0,Y 456.185,Z 460.126,A -85,B 0,C 180,E1 -8175.274,E2 -8175.274} C_VEL
LIN {X 0,Y 455.315,Z 470.83,A -85,B 0,C 180,E1 -8176.613,E2 -8176.613} C_VEL
LIN {X 0,Y 454.622,Z 479.672,A -85,B 0,C 180,E1 -8177.954,E2 -8177.954} C_VEL
LIN {X 0,Y 453.932,Z 488.13,A -85,B 0,C 180,E1 -8179.518,E2 -8179.518} C_VEL
LIN {X 0,Y 453.411,Z 494.975,A -85,B 0,C 180,E1 -8181.083,E2 -8181.083} C_VEL
LIN {X 0,Y 453.031,Z 501.134,A -85,B 0,C 180,E1 -8182.871,E2 -8182.871} C_VEL
LIN {X 0,Y 452.841,Z 504.712,A -85,B 0,C 180,E1 -8184.21,E2 -8184.21} C_VEL
LIN {X 0,Y 452.665,Z 507.5,A -85,B 0,C 180,E1 -8185.547,E2 -8185.547} C_VEL
LIN {X 0,Y 452.605,Z 510.03,A -85,B 0,C 180,E1 -8187.33,E2 -8187.33} C_VEL
LIN {X 0,Y 452.491,Z 511.299,A -85,B 0,C 180,E1 -8189.11,E2 -8189.11} C_VEL
LIN {X 0,Y 452.491,Z 511.332,A -85,B 0,C 180,E1 -8190.89,E2 -8190.89} C_VEL
LIN {X 0,Y 452.602,Z 510.136,A -85,B 0,C 180,E1 -8192.67,E2 -8192.67} C_VEL
LIN {X 0,Y 452.65,Z 507.678,A -85,B 0,C 180,E1 -8194.452,E2 -8194.452} C_VEL
LIN {X 0,Y 452.957,Z 503.859,A -85,B 0,C 180,E1 -8196.235,E2 -8196.235} C_VEL
LIN {X 0,Y 453.173,Z 498.584,A -85,B 0,C 180,E1 -8198.023,E2 -8198.023} C_VEL
LIN {X 0,Y 453.648,Z 491.659,A -85,B 0,C 180,E1 -8199.811,E2 -8199.811} C_VEL
LIN {X 0,Y 454.234,Z 484.021,A -85,B 0,C 180,E1 -8201.377,E2 -8201.377} C_VEL
LIN {X 0,Y 454.994,Z 474.942,A -85,B 0,C 180,E1 -8202.889,E2 -8202.889} C_VEL
LIN {X 0,Y 455.831,Z 464.711,A -85,B 0,C 180,E1 -8204.281,E2 -8204.281} C_VEL
LIN {X 0,Y 456.717,Z 453.653,A -85,B 0,C 180,E1 -8205.507,E2 -8205.507} C_VEL
LIN {X 0,Y 457.495,Z 442.68,A -85,B 0,C 180,E1 -8206.51,E2 -8206.51} C_VEL
LIN {X 0,Y 458.354,Z 430.719,A -85,B 0,C 180,E1 -8207.397,E2 -8207.397} C_VEL
LIN {X 0,Y 458.979,Z 419.139,A -85,B 0,C 180,E1 -8208.088,E2 -8208.088} C_VEL
LIN {X 0,Y 459.55,Z 405.081,A -85,B 0,C 180,E1 -8208.732,E2 -8208.732} C_VEL
LIN {X 0,Y 460.029,Z 391.159,A -85,B 0,C 180,E1 -8209.175,E2 -8209.175} C_VEL
LIN {X 0,Y 460.275,Z 376.906,A -85,B 0,C 180,E1 -8209.454,E2 -8209.454} C_VEL
LIN {X 0,Y 461.179,Z 265.591,A -85,B 0,C 180,E1 -8211.113,E2 -8211.113} C_VEL
LIN {X 0,Y 456.926,Z 244.461,A -85,B 0,C 180,E1 -8211.692,E2 -8211.692} C_VEL
LIN {X 0,Y 458.365,Z 220.988,A -85,B 0,C 180,E1 -8215.423,E2 -8215.423} C_VEL
LIN {X 0,Y 458.489,Z 216.591,A -85,B 0,C 180,E1 -8216.148,E2 -8216.148} C_VEL
LIN {X 0,Y 455.109,Z 202.022,A -85,B 0,C 180,E1 -8218.853,E2 -8218.853} C_VEL
LIN {X 0,Y 453.481,Z 195.676,A -85,B 0,C 180,E1 -8220.137,E2 -8220.137} C_VEL
LIN {X 0,Y 453.489,Z 195.603,A -85,B 0,C 180,E1 -8223.188,E2 -8223.188} C_VEL
LIN {X 0,Y 453.453,Z 195.621,A -85,B 0,C 180,E1 -8226.299,E2 -8226.299} C_VEL
LIN {X 0,Y 453.487,Z 195.618,A -85,B 0,C 180,E1 -8229.449,E2 -8229.449} C_VEL
LIN {X 0,Y 453.473,Z 195.617,A -85,B 0,C 180,E1 -8231.934,E2 -8231.934} C_VEL
LIN {X 0,Y 453.484,Z 195.617,A -85,B 0,C 180,E1 -8235.47,E2 -8235.47} C_VEL
LIN {X 0,Y 453.475,Z 195.622,A -85,B 0,C 180,E1 -8238.209,E2 -8238.209} C_VEL
LIN {X 0,Y 453.483,Z 195.612,A -85,B 0,C 180,E1 -8240.794,E2 -8240.794} C_VEL
LIN {X 0,Y 453.452,Z 195.62,A -85,B 0,C 180,E1 -8243.917,E2 -8243.917} C_VEL
LIN {X 0,Y 453.478,Z 195.62,A -85,B 0,C 180,E1 -8247.151,E2 -8247.151} C_VEL
LIN {X 0,Y 453.509,Z 195.609,A -85,B 0,C 180,E1 -8250.271,E2 -8250.271} C_VEL
LIN {X 0,Y 453.504,Z 195.618,A -85,B 0,C 180,E1 -8253.294,E2 -8253.294} C_VEL
LIN {X 0,Y 453.497,Z 195.615,A -85,B 0,C 180,E1 -8256.238,E2 -8256.238} C_VEL
LIN {X 0,Y 453.476,Z 195.621,A -85,B 0,C 180,E1 -8259.117,E2 -8259.117} C_VEL
LIN {X 0,Y 453.505,Z 195.616,A -85,B 0,C 180,E1 -8261.944,E2 -8261.944} C_VEL
LIN {X 0,Y 453.533,Z 195.613,A -85,B 0,C 180,E1 -8264.726,E2 -8264.726} C_VEL
LIN {X 0,Y 453.556,Z 195.607,A -85,B 0,C 180,E1 -8267.471,E2 -8267.471} C_VEL
LIN {X 0,Y 453.585,Z 195.606,A -85,B 0,C 180,E1 -8271.086,E2 -8271.086} C_VEL
LIN {X 0,Y 453.67,Z 195.595,A -85,B 0,C 180,E1 -8273.774,E2 -8273.774} C_VEL
LIN {X 0,Y 453.758,Z 195.581,A -85,B 0,C 180,E1 -8277.337,E2 -8277.337} C_VEL
LIN {X 0,Y 453.816,Z 195.58,A -85,B 0,C 180,E1 -8280,E2 -8280} C_VEL
LIN {X 0,Y 453.758,Z 195.588,A -85,B 0,C 180,E1 -8282.663,E2 -8282.663} C_VEL
LIN {X 0,Y 453.67,Z 195.596,A -85,B 0,C 180,E1 -8286.225,E2 -8286.225} C_VEL
LIN {X 0,Y 453.585,Z 195.604,A -85,B 0,C 180,E1 -8288.913,E2 -8288.913} C_VEL
LIN {X 0,Y 453.556,Z 195.61,A -85,B 0,C 180,E1 -8292.529,E2 -8292.529} C_VEL
LIN {X 0,Y 453.537,Z 195.615,A -85,B 0,C 180,E1 -8296.196,E2 -8296.196} C_VEL
LIN {X 0,Y 453.512,Z 195.614,A -85,B 0,C 180,E1 -8299.041,E2 -8299.041} C_VEL
LIN {X 0,Y 453.469,Z 195.622,A -85,B 0,C 180,E1 -8301.836,E2 -8301.836} C_VEL
LIN {X 0,Y 453.507,Z 195.612,A -85,B 0,C 180,E1 -8304.735,E2 -8304.735} C_VEL
LIN {X 0,Y 453.53,Z 195.61,A -85,B 0,C 180,E1 -8307.961,E2 -8307.961} C_VEL
LIN {X 0,Y 453.459,Z 195.617,A -85,B 0,C 180,E1 -8311.526,E2 -8311.526} C_VEL
LIN {X 0,Y 453.482,Z 195.62,A -85,B 0,C 180,E1 -8314.778,E2 -8314.778} C_VEL
LIN {X 0,Y 453.459,Z 195.619,A -85,B 0,C 180,E1 -8318.312,E2 -8318.312} C_VEL
LIN {X 0,Y 453.488,Z 195.62,A -85,B 0,C 180,E1 -8320.609,E2 -8320.609} C_VEL
LIN {X 0,Y 453.447,Z 195.625,A -85,B 0,C 180,E1 -8323.244,E2 -8323.244} C_VEL
LIN {X 0,Y 453.458,Z 195.62,A -85,B 0,C 180,E1 -8325.779,E2 -8325.779} C_VEL
LIN {X 0,Y 453.474,Z 195.619,A -85,B 0,C 180,E1 -8328.21,E2 -8328.21} C_VEL
LIN {X 0,Y 453.466,Z 195.6,A -85,B 0,C 180,E1 -8330.798,E2 -8330.798} C_VEL
LIN {X 0,Y 453.449,Z 195.614,A -85,B 0,C 180,E1 -8333.918,E2 -8333.918} C_VEL
LIN {X 0,Y 453.469,Z 195.618,A -85,B 0,C 180,E1 -8337.151,E2 -8337.151} C_VEL
LIN {X 0,Y 453.531,Z 195.846,A -85,B 0,C 180,E1 -8338.271,E2 -8338.271} C_VEL
LIN {X 0,Y 457.681,Z 211.039,A -85,B 0,C 180,E1 -8340.772,E2 -8340.772} C_VEL
LIN {X 0,Y 459.827,Z 219.849,A -85,B 0,C 180,E1 -8342.152,E2 -8342.152} C_VEL
LIN {X 0,Y 459.572,Z 225.626,A -85,B 0,C 180,E1 -8342.939,E2 -8342.939} C_VEL
LIN {X 0,Y 458.284,Z 245.224,A -85,B 0,C 180,E1 -8345.515,E2 -8345.515} C_VEL
LIN {X 0,Y 461.958,Z 267.799,A -85,B 0,C 180,E1 -8346.111,E2 -8346.111} C_VEL
LIN {X 0,Y 459.855,Z 408.922,A -85,B 0,C 180,E1 -8348.483,E2 -8348.483} C_VEL
LIN {X 0,Y 459.272,Z 424.521,A -85,B 0,C 180,E1 -8348.921,E2 -8348.921} C_VEL
LIN {X 0,Y 458.576,Z 439.698,A -85,B 0,C 180,E1 -8349.537,E2 -8349.537} C_VEL
LIN {X 0,Y 457.781,Z 453.399,A -85,B 0,C 180,E1 -8350.261,E2 -8350.261} C_VEL
LIN {X 0,Y 456.947,Z 466.886,A -85,B 0,C 180,E1 -8351.157,E2 -8351.157} C_VEL
LIN {X 0,Y 456.065,Z 480.625,A -85,B 0,C 180,E1 -8352.282,E2 -8352.282} C_VEL
LIN {X 0,Y 455.245,Z 492.819,A -85,B 0,C 180,E1 -8353.489,E2 -8353.489} C_VEL
LIN {X 0,Y 454.511,Z 503.594,A -85,B 0,C 180,E1 -8354.76,E2 -8354.76} C_VEL
LIN {X 0,Y 453.838,Z 514.815,A -85,B 0,C 180,E1 -8356.341,E2 -8356.341} C_VEL
LIN {X 0,Y 453.299,Z 524.819,A -85,B 0,C 180,E1 -8358.057,E2 -8358.057} C_VEL
LIN {X 0,Y 452.937,Z 532.807,A -85,B 0,C 180,E1 -8359.722,E2 -8359.722} C_VEL
LIN {X 0,Y 452.703,Z 539.778,A -85,B 0,C 180,E1 -8361.519,E2 -8361.519} C_VEL
LIN {X 0,Y 452.576,Z 545.348,A -85,B 0,C 180,E1 -8363.357,E2 -8363.357} C_VEL
LIN {X 0,Y 452.531,Z 548.376,A -85,B 0,C 180,E1 -8364.654,E2 -8364.654} C_VEL
LIN {X 0,Y 452.497,Z 551.464,A -85,B 0,C 180,E1 -8366.439,E2 -8366.439} C_VEL
LIN {X 0,Y 452.48,Z 553.306,A -85,B 0,C 180,E1 -8368.22,E2 -8368.22} C_VEL
LIN {X 0,Y 452.462,Z 553.932,A -85,B 0,C 180,E1 -8370,E2 -8370} C_VEL
LIN {X 0,Y 452.48,Z 553.302,A -85,B 0,C 180,E1 -8371.78,E2 -8371.78} C_VEL
LIN {X 0,Y 452.498,Z 551.457,A -85,B 0,C 180,E1 -8373.562,E2 -8373.562} C_VEL
LIN {X 0,Y 452.547,Z 548.372,A -85,B 0,C 180,E1 -8375.347,E2 -8375.347} C_VEL
LIN {X 0,Y 452.645,Z 543.976,A -85,B 0,C 180,E1 -8377.135,E2 -8377.135} C_VEL
LIN {X 0,Y 452.715,Z 538.152,A -85,B 0,C 180,E1 -8378.931,E2 -8378.931} C_VEL
LIN {X 0,Y 453.05,Z 530.759,A -85,B 0,C 180,E1 -8380.728,E2 -8380.728} C_VEL
LIN {X 0,Y 453.445,Z 521.964,A -85,B 0,C 180,E1 -8382.461,E2 -8382.461} C_VEL
LIN {X 0,Y 454.035,Z 511.764,A -85,B 0,C 180,E1 -8384.111,E2 -8384.111} C_VEL
LIN {X 0,Y 454.638,Z 501.749,A -85,B 0,C 180,E1 -8385.466,E2 -8385.466} C_VEL
LIN {X 0,Y 455.418,Z 490.187,A -85,B 0,C 180,E1 -8386.783,E2 -8386.783} C_VEL
LIN {X 0,Y 456.206,Z 478.004,A -85,B 0,C 180,E1 -8387.945,E2 -8387.945} C_VEL
LIN {X 0,Y 457.054,Z 465.242,A -85,B 0,C 180,E1 -8388.956,E2 -8388.956} C_VEL
LIN {X 0,Y 457.923,Z 451.362,A -85,B 0,C 180,E1 -8389.85,E2 -8389.85} C_VEL
LIN {X 0,Y 458.666,Z 437.162,A -85,B 0,C 180,E1 -8390.577,E2 -8390.577} C_VEL
LIN {X 0,Y 459.369,Z 422.591,A -85,B 0,C 180,E1 -8391.138,E2 -8391.138} C_VEL
LIN {X 0,Y 459.85,Z 407.375,A -85,B 0,C 180,E1 -8391.548,E2 -8391.548} C_VEL
LIN {X 0,Y 461.895,Z 267.822,A -85,B 0,C 180,E1 -8393.887,E2 -8393.887} C_VEL
LIN {X 0,Y 459.584,Z 253.076,A -85,B 0,C 180,E1 -8394.262,E2 -8394.262} C_VEL
LIN {X 0,Y 458.271,Z 245.111,A -85,B 0,C 180,E1 -8394.487,E2 -8394.487} C_VEL
LIN {X 0,Y 459.926,Z 221.679,A -85,B 0,C 180,E1 -8397.591,E2 -8397.591} C_VEL
LIN {X 0,Y 459.484,Z 218.295,A -85,B 0,C 180,E1 -8398.088,E2 -8398.088} C_VEL
LIN {X 0,Y 455.901,Z 204.258,A -85,B 0,C 180,E1 -8400.314,E2 -8400.314} C_VEL
LIN {X 0,Y 453.489,Z 195.729,A -85,B 0,C 180,E1 -8401.754,E2 -8401.754} C_VEL
LIN {X 0,Y 453.475,Z 195.604,A -85,B 0,C 180,E1 -8404.99,E2 -8404.99} C_VEL
LIN {X 0,Y 453.458,Z 195.617,A -85,B 0,C 180,E1 -8408.312,E2 -8408.312} C_VEL
LIN {X 0,Y 453.492,Z 195.597,A -85,B 0,C 180,E1 -8410.609,E2 -8410.609} C_VEL
LIN {X 0,Y 453.453,Z 195.624,A -85,B 0,C 180,E1 -8413.244,E2 -8413.244} C_VEL
LIN {X 0,Y 453.46,Z 195.623,A -85,B 0,C 180,E1 -8415.778,E2 -8415.778} C_VEL
LIN {X 0,Y 453.477,Z 195.615,A -85,B 0,C 180,E1 -8418.209,E2 -8418.209} C_VEL
LIN {X 0,Y 453.513,Z 195.617,A -85,B 0,C 180,E1 -8420.79,E2 -8420.79} C_VEL
LIN {X 0,Y 453.452,Z 195.623,A -85,B 0,C 180,E1 -8423.917,E2 -8423.917} C_VEL
LIN {X 0,Y 453.48,Z 195.607,A -85,B 0,C 180,E1 -8427.151,E2 -8427.151} C_VEL
LIN {X 0,Y 453.471,Z 195.626,A -85,B 0,C 180,E1 -8430.268,E2 -8430.268} C_VEL
LIN {X 0,Y 453.498,Z 195.601,A -85,B 0,C 180,E1 -8433.294,E2 -8433.294} C_VEL
LIN {X 0,Y 453.495,Z 195.623,A -85,B 0,C 180,E1 -8436.238,E2 -8436.238} C_VEL
LIN {X 0,Y 453.479,Z 195.617,A -85,B 0,C 180,E1 -8439.118,E2 -8439.118} C_VEL
LIN {X 0,Y 453.508,Z 195.617,A -85,B 0,C 180,E1 -8441.945,E2 -8441.945} C_VEL
LIN {X 0,Y 453.537,Z 195.612,A -85,B 0,C 180,E1 -8444.726,E2 -8444.726} C_VEL
LIN {X 0,Y 453.557,Z 195.612,A -85,B 0,C 180,E1 -8448.379,E2 -8448.379} C_VEL
LIN {X 0,Y 453.649,Z 195.604,A -85,B 0,C 180,E1 -8451.985,E2 -8451.985} C_VEL
LIN {X 0,Y 453.668,Z 195.591,A -85,B 0,C 180,E1 -8454.667,E2 -8454.667} C_VEL
LIN {X 0,Y 453.741,Z 195.59,A -85,B 0,C 180,E1 -8457.337,E2 -8457.337} C_VEL
LIN {X 0,Y 453.82,Z 195.58,A -85,B 0,C 180,E1 -8460,E2 -8460} C_VEL
LIN {X 0,Y 453.742,Z 195.583,A -85,B 0,C 180,E1 -8462.663,E2 -8462.663} C_VEL
LIN {X 0,Y 453.674,Z 195.594,A -85,B 0,C 180,E1 -8466.226,E2 -8466.226} C_VEL
LIN {X 0,Y 453.59,Z 195.605,A -85,B 0,C 180,E1 -8468.914,E2 -8468.914} C_VEL
LIN {X 0,Y 453.561,Z 195.606,A -85,B 0,C 180,E1 -8472.529,E2 -8472.529} C_VEL
LIN {X 0,Y 453.543,Z 195.607,A -85,B 0,C 180,E1 -8476.196,E2 -8476.196} C_VEL
LIN {X 0,Y 453.518,Z 195.618,A -85,B 0,C 180,E1 -8479.041,E2 -8479.041} C_VEL
LIN {X 0,Y 453.475,Z 195.621,A -85,B 0,C 180,E1 -8481.836,E2 -8481.836} C_VEL
LIN {X 0,Y 453.512,Z 195.617,A -85,B 0,C 180,E1 -8484.735,E2 -8484.735} C_VEL
LIN {X 0,Y 453.531,Z 195.603,A -85,B 0,C 180,E1 -8487.96,E2 -8487.96} C_VEL
LIN {X 0,Y 453.464,Z 195.623,A -85,B 0,C 180,E1 -8491.525,E2 -8491.525} C_VEL
LIN {X 0,Y 453.489,Z 195.61,A -85,B 0,C 180,E1 -8494.778,E2 -8494.778} C_VEL
LIN {X 0,Y 453.468,Z 195.625,A -85,B 0,C 180,E1 -8498.312,E2 -8498.312} C_VEL
LIN {X 0,Y 453.493,Z 195.613,A -85,B 0,C 180,E1 -8500.609,E2 -8500.609} C_VEL
LIN {X 0,Y 453.453,Z 195.62,A -85,B 0,C 180,E1 -8503.244,E2 -8503.244} C_VEL
LIN {X 0,Y 453.466,Z 195.622,A -85,B 0,C 180,E1 -8505.779,E2 -8505.779} C_VEL
LIN {X 0,Y 453.48,Z 195.617,A -85,B 0,C 180,E1 -8508.21,E2 -8508.21} C_VEL
LIN {X 0,Y 453.495,Z 195.616,A -85,B 0,C 180,E1 -8510.794,E2 -8510.794} C_VEL
LIN {X 0,Y 453.456,Z 195.622,A -85,B 0,C 180,E1 -8513.917,E2 -8513.917} C_VEL
LIN {X 0,Y 453.484,Z 195.605,A -85,B 0,C 180,E1 -8517.151,E2 -8517.151} C_VEL
LIN {X 0,Y 453.506,Z 195.786,A -85,B 0,C 180,E1 -8520.023,E2 -8520.023} C_VEL
LIN {X 0,Y 456.723,Z 208.721,A -85,B 0,C 180,E1 -8522.507,E2 -8522.507} C_VEL
LIN {X 0,Y 458.574,Z 217.434,A -85,B 0,C 180,E1 -8524.101,E2 -8524.101} C_VEL
LIN {X 0,Y 457.223,Z 237.955,A -85,B 0,C 180,E1 -8527.401,E2 -8527.401} C_VEL
LIN {X 0,Y 456.906,Z 244.625,A -85,B 0,C 180,E1 -8528.412,E2 -8528.412} C_VEL
LIN {X 0,Y 461.252,Z 266.603,A -85,B 0,C 180,E1 -8529,E2 -8529} C_VEL
LIN {X 0,Y 460.758,Z 329.041,A -85,B 0,C 180,E1 -8529.936,E2 -8529.936} C_VEL
LIN {X 0,Y 460.102,Z 334.895,A -85,B 0,C 180,E1 -8529.993,E2 -8529.993} C_VEL
LIN {X 0,Y 454.477,Z 353.937,A -85,B 0,C 180,E1 -8530.007,E2 -8530.007} C_VEL
LIN {X 0,Y 453.809,Z 359.792,A -85,B 0,C 180,E1 -8530.064,E2 -8530.064} C_VEL
LIN {X 0,Y 453.479,Z 387.239,A -85,B 0,C 180,E1 -8530.507,E2 -8530.507} C_VEL
LIN {X 0,Y 453.085,Z 401.05,A -85,B 0,C 180,E1 -8530.901,E2 -8530.901} C_VEL
LIN {X 0,Y 452.529,Z 415.076,A -85,B 0,C 180,E1 -8531.493,E2 -8531.493} C_VEL
LIN {X 0,Y 451.948,Z 426.317,A -85,B 0,C 180,E1 -8532.114,E2 -8532.114} C_VEL
LIN {X 0,Y 451.039,Z 439.203,A -85,B 0,C 180,E1 -8533.013,E2 -8533.013} C_VEL
LIN {X 0,Y 450.135,Z 450.862,A -85,B 0,C 180,E1 -8534.027,E2 -8534.027} C_VEL
LIN {X 0,Y 449.162,Z 462.463,A -85,B 0,C 180,E1 -8535.27,E2 -8535.27} C_VEL
LIN {X 0,Y 448.33,Z 472.426,A -85,B 0,C 180,E1 -8536.574,E2 -8536.574} C_VEL
LIN {X 0,Y 447.562,Z 481.375,A -85,B 0,C 180,E1 -8537.991,E2 -8537.991} C_VEL
LIN {X 0,Y 446.873,Z 489.583,A -85,B 0,C 180,E1 -8539.58,E2 -8539.58} C_VEL
LIN {X 0,Y 446.396,Z 495.336,A -85,B 0,C 180,E1 -8540.942,E2 -8540.942} C_VEL
LIN {X 0,Y 445.984,Z 501.485,A -85,B 0,C 180,E1 -8542.757,E2 -8542.757} C_VEL
LIN {X 0,Y 445.802,Z 505.055,A -85,B 0,C 180,E1 -8544.118,E2 -8544.118} C_VEL
LIN {X 0,Y 445.58,Z 507.841,A -85,B 0,C 180,E1 -8545.476,E2 -8545.476} C_VEL
LIN {X 0,Y 445.53,Z 510.366,A -85,B 0,C 180,E1 -8547.287,E2 -8547.287} C_VEL
LIN {X 0,Y 445.413,Z 511.631,A -85,B 0,C 180,E1 -8549.096,E2 -8549.096} C_VEL
LIN {X 0,Y 445.412,Z 511.664,A -85,B 0,C 180,E1 -8550.904,E2 -8550.904} C_VEL
LIN {X 0,Y 445.527,Z 510.47,A -85,B 0,C 180,E1 -8552.712,E2 -8552.712} C_VEL
LIN {X 0,Y 445.566,Z 508.017,A -85,B 0,C 180,E1 -8554.523,E2 -8554.523} C_VEL
LIN {X 0,Y 445.892,Z 504.205,A -85,B 0,C 180,E1 -8556.334,E2 -8556.334} C_VEL
LIN {X 0,Y 446.125,Z 498.937,A -85,B 0,C 180,E1 -8558.15,E2 -8558.15} C_VEL
LIN {X 0,Y 446.652,Z 492.021,A -85,B 0,C 180,E1 -8559.967,E2 -8559.967} C_VEL
LIN {X 0,Y 447.273,Z 484.396,A -85,B 0,C 180,E1 -8561.556,E2 -8561.556} C_VEL
LIN {X 0,Y 448.059,Z 475.535,A -85,B 0,C 180,E1 -8563.06,E2 -8563.06} C_VEL
LIN {X 0,Y 448.958,Z 465.121,A -85,B 0,C 180,E1 -8564.504,E2 -8564.504} C_VEL
LIN {X 0,Y 449.875,Z 454.1,A -85,B 0,C 180,E1 -8565.749,E2 -8565.749} C_VEL
LIN {X 0,Y 450.721,Z 443.157,A -85,B 0,C 180,E1 -8566.766,E2 -8566.766} C_VEL
LIN {X 0,Y 451.611,Z 431.249,A -85,B 0,C 180,E1 -8567.665,E2 -8567.665} C_VEL
LIN {X 0,Y 452.336,Z 418.625,A -85,B 0,C 180,E1 -8568.425,E2 -8568.425} C_VEL
LIN {X 0,Y 452.944,Z 404.296,A -85,B 0,C 180,E1 -8569.075,E2 -8569.075} C_VEL
LIN {X 0,Y 453.418,Z 391.021,A -85,B 0,C 180,E1 -8569.495,E2 -8569.495} C_VEL
LIN {X 0,Y 453.665,Z 376.552,A -85,B 0,C 180,E1 -8569.778,E2 -8569.778} C_VEL
LIN {X 0,Y 454.671,Z 266.915,A -85,B 0,C 180,E1 -8571.433,E2 -8571.433} C_VEL
LIN {X 0,Y 450.144,Z 244.415,A -85,B 0,C 180,E1 -8572.065,E2 -8572.065} C_VEL
LIN {X 0,Y 451.559,Z 222.72,A -85,B 0,C 180,E1 -8575.563,E2 -8575.563} C_VEL
LIN {X 0,Y 451.657,Z 218.184,A -85,B 0,C 180,E1 -8576.325,E2 -8576.325} C_VEL
LIN {X 0,Y 448.236,Z 203.583,A -85,B 0,C 180,E1 -8579.081,E2 -8579.081} C_VEL
LIN {X 0,Y 446.438,Z 196.572,A -85,B 0,C 180,E1 -8580.509,E2 -8580.509} C_VEL
LIN {X 0,Y 446.444,Z 196.48,A -85,B 0,C 180,E1 -8583.453,E2 -8583.453} C_VEL
LIN {X 0,Y 446.407,Z 196.499,A -85,B 0,C 180,E1 -8586.744,E2 -8586.744} C_VEL
LIN {X 0,Y 446.452,Z 196.495,A -85,B 0,C 180,E1 -8589.524,E2 -8589.524} C_VEL
LIN {X 0,Y 446.426,Z 196.494,A -85,B 0,C 180,E1 -8592.604,E2 -8592.604} C_VEL
LIN {X 0,Y 446.45,Z 196.496,A -85,B 0,C 180,E1 -8595.103,E2 -8595.103} C_VEL
LIN {X 0,Y 446.424,Z 196.5,A -85,B 0,C 180,E1 -8598.608,E2 -8598.608} C_VEL
LIN {X 0,Y 446.435,Z 196.491,A -85,B 0,C 180,E1 -8600.972,E2 -8600.972} C_VEL
LIN {X 0,Y 446.417,Z 196.495,A -85,B 0,C 180,E1 -8604.373,E2 -8604.373} C_VEL
LIN {X 0,Y 446.417,Z 196.503,A -85,B 0,C 180,E1 -8607.638,E2 -8607.638} C_VEL
LIN {X 0,Y 446.464,Z 196.483,A -85,B 0,C 180,E1 -8610.792,E2 -8610.792} C_VEL
LIN {X 0,Y 446.472,Z 196.492,A -85,B 0,C 180,E1 -8613.848,E2 -8613.848} C_VEL
LIN {X 0,Y 446.423,Z 196.499,A -85,B 0,C 180,E1 -8616.823,E2 -8616.823} C_VEL
LIN {X 0,Y 446.437,Z 196.492,A -85,B 0,C 180,E1 -8619.737,E2 -8619.737} C_VEL
LIN {X 0,Y 446.457,Z 196.499,A -85,B 0,C 180,E1 -8622.597,E2 -8622.597} C_VEL
LIN {X 0,Y 446.466,Z 196.494,A -85,B 0,C 180,E1 -8625.412,E2 -8625.412} C_VEL
LIN {X 0,Y 446.511,Z 196.486,A -85,B 0,C 180,E1 -8628.193,E2 -8628.193} C_VEL
LIN {X 0,Y 446.593,Z 196.475,A -85,B 0,C 180,E1 -8631.858,E2 -8631.858} C_VEL
LIN {X 0,Y 446.639,Z 196.478,A -85,B 0,C 180,E1 -8634.582,E2 -8634.582} C_VEL
LIN {X 0,Y 446.702,Z 196.46,A -85,B 0,C 180,E1 -8637.295,E2 -8637.295} C_VEL
LIN {X 0,Y 446.786,Z 196.456,A -85,B 0,C 180,E1 -8640,E2 -8640} C_VEL
LIN {X 0,Y 446.702,Z 196.467,A -85,B 0,C 180,E1 -8642.705,E2 -8642.705} C_VEL
LIN {X 0,Y 446.639,Z 196.473,A -85,B 0,C 180,E1 -8646.324,E2 -8646.324} C_VEL
LIN {X 0,Y 446.531,Z 196.482,A -85,B 0,C 180,E1 -8649.055,E2 -8649.055} C_VEL
LIN {X 0,Y 446.514,Z 196.486,A -85,B 0,C 180,E1 -8652.73,E2 -8652.73} C_VEL
LIN {X 0,Y 446.489,Z 196.493,A -85,B 0,C 180,E1 -8656.228,E2 -8656.228} C_VEL
LIN {X 0,Y 446.462,Z 196.494,A -85,B 0,C 180,E1 -8659.303,E2 -8659.303} C_VEL
LIN {X 0,Y 446.411,Z 196.504,A -85,B 0,C 180,E1 -8662.2,E2 -8662.2} C_VEL
LIN {X 0,Y 446.452,Z 196.492,A -85,B 0,C 180,E1 -8665.152,E2 -8665.152} C_VEL
LIN {X 0,Y 446.478,Z 196.493,A -85,B 0,C 180,E1 -8668.179,E2 -8668.179} C_VEL
LIN {X 0,Y 446.412,Z 196.49,A -85,B 0,C 180,E1 -8671.775,E2 -8671.775} C_VEL
LIN {X 0,Y 446.424,Z 196.499,A -85,B 0,C 180,E1 -8674.523,E2 -8674.523} C_VEL
LIN {X 0,Y 446.41,Z 196.496,A -85,B 0,C 180,E1 -8678.08,E2 -8678.08} C_VEL
LIN {X 0,Y 446.421,Z 196.502,A -85,B 0,C 180,E1 -8680.918,E2 -8680.918} C_VEL
LIN {X 0,Y 446.393,Z 196.505,A -85,B 0,C 180,E1 -8683.847,E2 -8683.847} C_VEL
LIN {X 0,Y 446.393,Z 196.502,A -85,B 0,C 180,E1 -8686.404,E2 -8686.404} C_VEL
LIN {X 0,Y 446.422,Z 196.481,A -85,B 0,C 180,E1 -8689.083,E2 -8689.083} C_VEL
LIN {X 0,Y 446.403,Z 196.503,A -85,B 0,C 180,E1 -8692.122,E2 -8692.122} C_VEL
LIN {X 0,Y 446.418,Z 196.485,A -85,B 0,C 180,E1 -8695.477,E2 -8695.477} C_VEL
LIN {X 0,Y 446.471,Z 196.678,A -85,B 0,C 180,E1 -8697.849,E2 -8697.849} C_VEL
LIN {X 0,Y 450.812,Z 212.42,A -85,B 0,C 180,E1 -8700.504,E2 -8700.504} C_VEL
LIN {X 0,Y 453.158,Z 222.686,A -85,B 0,C 180,E1 -8702.13,E2 -8702.13} C_VEL
LIN {X 0,Y 451.588,Z 245.229,A -85,B 0,C 180,E1 -8705.154,E2 -8705.154} C_VEL
LIN {X 0,Y 455.334,Z 267.723,A -85,B 0,C 180,E1 -8705.765,E2 -8705.765} C_VEL
LIN {X 0,Y 453.206,Z 407.762,A -85,B 0,C 180,E1 -8708.151,E2 -8708.151} C_VEL
LIN {X 0,Y 452.604,Z 423.315,A -85,B 0,C 180,E1 -8708.581,E2 -8708.581} C_VEL
LIN {X 0,Y 451.879,Z 439.069,A -85,B 0,C 180,E1 -8709.22,E2 -8709.22} C_VEL
LIN {X 0,Y 451.05,Z 452.831,A -85,B 0,C 180,E1 -8709.954,E2 -8709.954} C_VEL
LIN {X 0,Y 450.155,Z 466.365,A -85,B 0,C 180,E1 -8710.862,E2 -8710.862} C_VEL
LIN {X 0,Y 449.194,Z 480.157,A -85,B 0,C 180,E1 -8712.001,E2 -8712.001} C_VEL
LIN {X 0,Y 448.321,Z 492.824,A -85,B 0,C 180,E1 -8713.278,E2 -8713.278} C_VEL
LIN {X 0,Y 447.442,Z 504.903,A -85,B 0,C 180,E1 -8714.747,E2 -8714.747} C_VEL
LIN {X 0,Y 446.867,Z 514.418,A -85,B 0,C 180,E1 -8716.123,E2 -8716.123} C_VEL
LIN {X 0,Y 446.269,Z 523.402,A -85,B 0,C 180,E1 -8717.666,E2 -8717.666} C_VEL
LIN {X 0,Y 445.97,Z 531.445,A -85,B 0,C 180,E1 -8719.33,E2 -8719.33} C_VEL
LIN {X 0,Y 445.638,Z 537.799,A -85,B 0,C 180,E1 -8720.927,E2 -8720.927} C_VEL
LIN {X 0,Y 445.503,Z 543.624,A -85,B 0,C 180,E1 -8722.75,E2 -8722.75} C_VEL
LIN {X 0,Y 445.443,Z 548.034,A -85,B 0,C 180,E1 -8724.568,E2 -8724.568} C_VEL
LIN {X 0,Y 445.396,Z 551.127,A -85,B 0,C 180,E1 -8726.382,E2 -8726.382} C_VEL
LIN {X 0,Y 445.396,Z 552.973,A -85,B 0,C 180,E1 -8728.192,E2 -8728.192} C_VEL
LIN {X 0,Y 445.398,Z 553.6,A -85,B 0,C 180,E1 -8730,E2 -8730} C_VEL
LIN {X 0,Y 445.396,Z 552.969,A -85,B 0,C 180,E1 -8731.809,E2 -8731.809} C_VEL
LIN {X 0,Y 445.396,Z 551.119,A -85,B 0,C 180,E1 -8733.619,E2 -8733.619} C_VEL
LIN {X 0,Y 445.461,Z 548.028,A -85,B 0,C 180,E1 -8735.432,E2 -8735.432} C_VEL
LIN {X 0,Y 445.566,Z 543.624,A -85,B 0,C 180,E1 -8737.249,E2 -8737.249} C_VEL
LIN {X 0,Y 445.639,Z 537.789,A -85,B 0,C 180,E1 -8739.074,E2 -8739.074} C_VEL
LIN {X 0,Y 446.01,Z 530.385,A -85,B 0,C 180,E1 -8740.9,E2 -8740.9} C_VEL
LIN {X 0,Y 446.394,Z 522.205,A -85,B 0,C 180,E1 -8742.546,E2 -8742.546} C_VEL
LIN {X 0,Y 446.972,Z 512.883,A -85,B 0,C 180,E1 -8744.106,E2 -8744.106} C_VEL
LIN {X 0,Y 447.561,Z 503.144,A -85,B 0,C 180,E1 -8745.483,E2 -8745.483} C_VEL
LIN {X 0,Y 448.37,Z 491.755,A -85,B 0,C 180,E1 -8746.837,E2 -8746.837} C_VEL
LIN {X 0,Y 449.276,Z 478.829,A -85,B 0,C 180,E1 -8748.114,E2 -8748.114} C_VEL
LIN {X 0,Y 450.162,Z 466.309,A -85,B 0,C 180,E1 -8749.139,E2 -8749.139} C_VEL
LIN {X 0,Y 451.059,Z 452.755,A -85,B 0,C 180,E1 -8750.047,E2 -8750.047} C_VEL
LIN {X 0,Y 451.917,Z 437.758,A -85,B 0,C 180,E1 -8750.839,E2 -8750.839} C_VEL
LIN {X 0,Y 452.665,Z 422.752,A -85,B 0,C 180,E1 -8751.432,E2 -8751.432} C_VEL
LIN {X 0,Y 453.193,Z 407.546,A -85,B 0,C 180,E1 -8751.85,E2 -8751.85} C_VEL
LIN {X 0,Y 455.314,Z 271.493,A -85,B 0,C 180,E1 -8754.164,E2 -8754.164} C_VEL
LIN {X 0,Y 455.085,Z 266.262,A -85,B 0,C 180,E1 -8754.268,E2 -8754.268} C_VEL
LIN {X 0,Y 451.552,Z 245.111,A -85,B 0,C 180,E1 -8754.849,E2 -8754.849} C_VEL
LIN {X 0,Y 453.16,Z 222.707,A -85,B 0,C 180,E1 -8757.871,E2 -8757.871} C_VEL
LIN {X 0,Y 450.442,Z 210.893,A -85,B 0,C 180,E1 -8759.738,E2 -8759.738} C_VEL
LIN {X 0,Y 446.457,Z 196.583,A -85,B 0,C 180,E1 -8762.173,E2 -8762.173} C_VEL
LIN {X 0,Y 446.416,Z 196.484,A -85,B 0,C 180,E1 -8765.626,E2 -8765.626} C_VEL
LIN {X 0,Y 446.424,Z 196.477,A -85,B 0,C 180,E1 -8769.029,E2 -8769.029} C_VEL
LIN {X 0,Y 446.433,Z 196.499,A -85,B 0,C 180,E1 -8772.277,E2 -8772.277} C_VEL
LIN {X 0,Y 446.449,Z 196.497,A -85,B 0,C 180,E1 -8775.104,E2 -8775.104} C_VEL
LIN {X 0,Y 446.426,Z 196.495,A -85,B 0,C 180,E1 -8778.609,E2 -8778.609} C_VEL
LIN {X 0,Y 446.457,Z 196.494,A -85,B 0,C 180,E1 -8780.974,E2 -8780.974} C_VEL
LIN {X 0,Y 446.417,Z 196.504,A -85,B 0,C 180,E1 -8784.374,E2 -8784.374} C_VEL
LIN {X 0,Y 446.419,Z 196.486,A -85,B 0,C 180,E1 -8787.638,E2 -8787.638} C_VEL
LIN {X 0,Y 446.445,Z 196.497,A -85,B 0,C 180,E1 -8790.791,E2 -8790.791} C_VEL
LIN {X 0,Y 446.475,Z 196.476,A -85,B 0,C 180,E1 -8793.848,E2 -8793.848} C_VEL
LIN {X 0,Y 446.423,Z 196.5,A -85,B 0,C 180,E1 -8796.823,E2 -8796.823} C_VEL
LIN {X 0,Y 446.441,Z 196.497,A -85,B 0,C 180,E1 -8799.737,E2 -8799.737} C_VEL
LIN {X 0,Y 446.46,Z 196.494,A -85,B 0,C 180,E1 -8802.597,E2 -8802.597} C_VEL
LIN {X 0,Y 446.467,Z 196.493,A -85,B 0,C 180,E1 -8805.412,E2 -8805.412} C_VEL
LIN {X 0,Y 446.515,Z 196.491,A -85,B 0,C 180,E1 -8808.193,E2 -8808.193} C_VEL
LIN {X 0,Y 446.598,Z 196.482,A -85,B 0,C 180,E1 -8811.858,E2 -8811.858} C_VEL
LIN {X 0,Y 446.642,Z 196.466,A -85,B 0,C 180,E1 -8814.583,E2 -8814.583} C_VEL
LIN {X 0,Y 446.661,Z 196.465,A -85,B 0,C 180,E1 -8818.197,E2 -8818.197} C_VEL
LIN {X 0,Y 446.79,Z 196.456,A -85,B 0,C 180,E1 -8820,E2 -8820} C_VEL
LIN {X 0,Y 446.689,Z 196.462,A -85,B 0,C 180,E1 -8822.706,E2 -8822.706} C_VEL
LIN {X 0,Y 446.644,Z 196.469,A -85,B 0,C 180,E1 -8826.324,E2 -8826.324} C_VEL
LIN {X 0,Y 446.536,Z 196.485,A -85,B 0,C 180,E1 -8829.056,E2 -8829.056} C_VEL
LIN {X 0,Y 446.52,Z 196.484,A -85,B 0,C 180,E1 -8832.73,E2 -8832.73} C_VEL
LIN {X 0,Y 446.494,Z 196.485,A -85,B 0,C 180,E1 -8836.228,E2 -8836.228} C_VEL
LIN {X 0,Y 446.467,Z 196.493,A -85,B 0,C 180,E1 -8839.303,E2 -8839.303} C_VEL
LIN {X 0,Y 446.416,Z 196.5,A -85,B 0,C 180,E1 -8842.2,E2 -8842.2} C_VEL
LIN {X 0,Y 446.456,Z 196.5,A -85,B 0,C 180,E1 -8845.153,E2 -8845.153} C_VEL
LIN {X 0,Y 446.483,Z 196.481,A -85,B 0,C 180,E1 -8848.179,E2 -8848.179} C_VEL
LIN {X 0,Y 446.418,Z 196.5,A -85,B 0,C 180,E1 -8851.775,E2 -8851.775} C_VEL
LIN {X 0,Y 446.43,Z 196.489,A -85,B 0,C 180,E1 -8854.523,E2 -8854.523} C_VEL
LIN {X 0,Y 446.428,Z 196.5,A -85,B 0,C 180,E1 -8858.082,E2 -8858.082} C_VEL
LIN {X 0,Y 446.427,Z 196.498,A -85,B 0,C 180,E1 -8860.918,E2 -8860.918} C_VEL
LIN {X 0,Y 446.4,Z 196.498,A -85,B 0,C 180,E1 -8863.846,E2 -8863.846} C_VEL
LIN {X 0,Y 446.416,Z 196.505,A -85,B 0,C 180,E1 -8866.401,E2 -8866.401} C_VEL
LIN {X 0,Y 446.444,Z 196.5,A -85,B 0,C 180,E1 -8869.802,E2 -8869.802} C_VEL
LIN {X 0,Y 446.428,Z 196.502,A -85,B 0,C 180,E1 -8872.123,E2 -8872.123} C_VEL
LIN {X 0,Y 446.431,Z 196.496,A -85,B 0,C 180,E1 -8875.477,E2 -8875.477} C_VEL
LIN {X 0,Y 446.418,Z 196.504,A -85,B 0,C 180,E1 -8878.7,E2 -8878.7} C_VEL
LIN {X 0,Y 446.47,Z 196.733,A -85,B 0,C 180,E1 -8879.656,E2 -8879.656} C_VEL
LIN {X 0,Y 449.851,Z 210.126,A -85,B 0,C 180,E1 -8882.273,E2 -8882.273} C_VEL
LIN {X 0,Y 451.773,Z 219.027,A -85,B 0,C 180,E1 -8883.93,E2 -8883.93} C_VEL
LIN {X 0,Y 450.409,Z 238.923,A -85,B 0,C 180,E1 -8887.174,E2 -8887.174} C_VEL
LIN {X 0,Y 450.11,Z 244.335,A -85,B 0,C 180,E1 -8888.021,E2 -8888.021} C_VEL
LIN {X 0,Y 452.688,Z 257.063,A -85,B 0,C 180,E1 -8888.398,E2 -8888.398} C_VEL
LIN {X 0,Y 454.694,Z 267.499,A -85,B 0,C 180,E1 -8888.671,E2 -8888.671} C_VEL
LIN {X 0,Y 453.809,Z 359.792,A -85,B 0,C 180,E1 -8890.064,E2 -8890.064} C_VEL
LIN {X 0,Y 453.163,Z 365.647,A -85,B 0,C 180,E1 -8890.12,E2 -8890.12} C_VEL
LIN {X 0,Y 447.558,Z 384.675,A -85,B 0,C 180,E1 -8890.157,E2 -8890.157} C_VEL
LIN {X 0,Y 446.806,Z 390.481,A -85,B 0,C 180,E1 -8890.259,E2 -8890.259} C_VEL
LIN {X 0,Y 446.341,Z 404.136,A -85,B 0,C 180,E1 -8890.691,E2 -8890.691} C_VEL
LIN {X 0,Y 445.688,Z 417.854,A -85,B 0,C 180,E1 -8891.311,E2 -8891.311} C_VEL
LIN {X 0,Y 444.998,Z 430.369,A -85,B 0,C 180,E1 -8892.063,E2 -8892.063} C_VEL
LIN {X 0,Y 444.052,Z 442.512,A -85,B 0,C 180,E1 -8892.974,E2 -8892.974} C_VEL
LIN {X 0,Y 443.121,Z 453.62,A -85,B 0,C 180,E1 -8894.004,E2 -8894.004} C_VEL
LIN {X 0,Y 442.143,Z 464.794,A -85,B 0,C 180,E1 -8895.266,E2 -8895.266} C_VEL
LIN {X 0,Y 441.316,Z 474.258,A -85,B 0,C 180,E1 -8896.568,E2 -8896.568} C_VEL
LIN {X 0,Y 440.478,Z 483.071,A -85,B 0,C 180,E1 -8898.029,E2 -8898.029} C_VEL
LIN {X 0,Y 439.826,Z 491.001,A -85,B 0,C 180,E1 -8899.644,E2 -8899.644} C_VEL
LIN {X 0,Y 439.261,Z 497.414,A -85,B 0,C 180,E1 -8901.257,E2 -8901.257} C_VEL
LIN {X 0,Y 438.88,Z 503.215,A -85,B 0,C 180,E1 -8903.14,E2 -8903.14} C_VEL
LIN {X 0,Y 438.617,Z 506.422,A -85,B 0,C 180,E1 -8904.483,E2 -8904.483} C_VEL
LIN {X 0,Y 438.555,Z 509.599,A -85,B 0,C 180,E1 -8906.324,E2 -8906.324} C_VEL
LIN {X 0,Y 438.376,Z 511.488,A -85,B 0,C 180,E1 -8908.162,E2 -8908.162} C_VEL
LIN {X 0,Y 438.314,Z 512.133,A -85,B 0,C 180,E1 -8910,E2 -8910} C_VEL
LIN {X 0,Y 438.362,Z 511.555,A -85,B 0,C 180,E1 -8911.837,E2 -8911.837} C_VEL
LIN {X 0,Y 438.545,Z 509.737,A -85,B 0,C 180,E1 -8913.675,E2 -8913.675} C_VEL
LIN {X 0,Y 438.615,Z 506.629,A -85,B 0,C 180,E1 -8915.516,E2 -8915.516} C_VEL
LIN {X 0,Y 438.878,Z 503.457,A -85,B 0,C 180,E1 -8916.858,E2 -8916.858} C_VEL
LIN {X 0,Y 439.212,Z 497.734,A -85,B 0,C 180,E1 -8918.743,E2 -8918.743} C_VEL
LIN {X 0,Y 439.642,Z 492.381,A -85,B 0,C 180,E1 -8920.127,E2 -8920.127} C_VEL
LIN {X 0,Y 440.322,Z 484.766,A -85,B 0,C 180,E1 -8921.741,E2 -8921.741} C_VEL
LIN {X 0,Y 441.137,Z 476.083,A -85,B 0,C 180,E1 -8923.242,E2 -8923.242} C_VEL
LIN {X 0,Y 441.91,Z 467.268,A -85,B 0,C 180,E1 -8924.506,E2 -8924.506} C_VEL
LIN {X 0,Y 442.885,Z 456.656,A -85,B 0,C 180,E1 -8925.768,E2 -8925.768} C_VEL
LIN {X 0,Y 443.724,Z 446.177,A -85,B 0,C 180,E1 -8926.801,E2 -8926.801} C_VEL
LIN {X 0,Y 444.607,Z 434.908,A -85,B 0,C 180,E1 -8927.715,E2 -8927.715} C_VEL
LIN {X 0,Y 445.439,Z 422.139,A -85,B 0,C 180,E1 -8928.546,E2 -8928.546} C_VEL
LIN {X 0,Y 446.131,Z 408.303,A -85,B 0,C 180,E1 -8929.236,E2 -8929.236} C_VEL
LIN {X 0,Y 446.691,Z 394.067,A -85,B 0,C 180,E1 -8929.741,E2 -8929.741} C_VEL
LIN {X 0,Y 446.994,Z 379.905,A -85,B 0,C 180,E1 -8930.056,E2 -8930.056} C_VEL
LIN {X 0,Y 448.126,Z 267.875,A -85,B 0,C 180,E1 -8931.771,E2 -8931.771} C_VEL
LIN {X 0,Y 443.409,Z 244.506,A -85,B 0,C 180,E1 -8932.437,E2 -8932.437} C_VEL
LIN {X 0,Y 444.855,Z 223.224,A -85,B 0,C 180,E1 -8935.912,E2 -8935.912} C_VEL
LIN {X 0,Y 444.811,Z 219.776,A -85,B 0,C 180,E1 -8936.509,E2 -8936.509} C_VEL
LIN {X 0,Y 441.558,Z 205.868,A -85,B 0,C 180,E1 -8939.173,E2 -8939.173} C_VEL
LIN {X 0,Y 439.411,Z 197.442,A -85,B 0,C 180,E1 -8940.917,E2 -8940.917} C_VEL
LIN {X 0,Y 439.386,Z 197.362,A -85,B 0,C 180,E1 -8944.043,E2 -8944.043} C_VEL
LIN {X 0,Y 439.355,Z 197.377,A -85,B 0,C 180,E1 -8946.888,E2 -8946.888} C_VEL
LIN {X 0,Y 439.399,Z 197.375,A -85,B 0,C 180,E1 -8949.848,E2 -8949.848} C_VEL
LIN {X 0,Y 439.379,Z 197.371,A -85,B 0,C 180,E1 -8952.626,E2 -8952.626} C_VEL
LIN {X 0,Y 439.398,Z 197.372,A -85,B 0,C 180,E1 -8955.27,E2 -8955.27} C_VEL
LIN {X 0,Y 439.384,Z 197.378,A -85,B 0,C 180,E1 -8958.742,E2 -8958.742} C_VEL
LIN {X 0,Y 439.375,Z 197.379,A -85,B 0,C 180,E1 -8961.606,E2 -8961.606} C_VEL
LIN {X 0,Y 439.396,Z 197.367,A -85,B 0,C 180,E1 -8964.843,E2 -8964.843} C_VEL
LIN {X 0,Y 439.369,Z 197.378,A -85,B 0,C 180,E1 -8968.139,E2 -8968.139} C_VEL
LIN {X 0,Y 439.42,Z 197.357,A -85,B 0,C 180,E1 -8971.326,E2 -8971.326} C_VEL
LIN {X 0,Y 439.399,Z 197.374,A -85,B 0,C 180,E1 -8974.415,E2 -8974.415} C_VEL
LIN {X 0,Y 439.359,Z 197.381,A -85,B 0,C 180,E1 -8977.424,E2 -8977.424} C_VEL
LIN {X 0,Y 439.435,Z 197.368,A -85,B 0,C 180,E1 -8980.662,E2 -8980.662} C_VEL
LIN {X 0,Y 439.456,Z 197.363,A -85,B 0,C 180,E1 -8984.224,E2 -8984.224} C_VEL
LIN {X 0,Y 439.477,Z 197.361,A -85,B 0,C 180,E1 -8987.285,E2 -8987.285} C_VEL
LIN {X 0,Y 439.493,Z 197.365,A -85,B 0,C 180,E1 -8990.798,E2 -8990.798} C_VEL
LIN {X 0,Y 439.611,Z 197.346,A -85,B 0,C 180,E1 -8993.575,E2 -8993.575} C_VEL
LIN {X 0,Y 439.649,Z 197.339,A -85,B 0,C 180,E1 -8997.251,E2 -8997.251} C_VEL
LIN {X 0,Y 439.756,Z 197.331,A -85,B 0,C 180,E1 -9000,E2 -9000} C_VEL
LIN {X 0,Y 439.649,Z 197.345,A -85,B 0,C 180,E1 -9002.749,E2 -9002.749} C_VEL
LIN {X 0,Y 439.611,Z 197.35,A -85,B 0,C 180,E1 -9006.425,E2 -9006.425} C_VEL
LIN {X 0,Y 439.492,Z 197.359,A -85,B 0,C 180,E1 -9009.202,E2 -9009.202} C_VEL
LIN {X 0,Y 439.458,Z 197.364,A -85,B 0,C 180,E1 -9012.938,E2 -9012.938} C_VEL
LIN {X 0,Y 439.44,Z 197.37,A -85,B 0,C 180,E1 -9016.349,E2 -9016.349} C_VEL
LIN {X 0,Y 439.395,Z 197.377,A -85,B 0,C 180,E1 -9019.626,E2 -9019.626} C_VEL
LIN {X 0,Y 439.358,Z 197.379,A -85,B 0,C 180,E1 -9022.576,E2 -9022.576} C_VEL
LIN {X 0,Y 439.399,Z 197.364,A -85,B 0,C 180,E1 -9025.585,E2 -9025.585} C_VEL
LIN {X 0,Y 439.41,Z 197.371,A -85,B 0,C 180,E1 -9028.674,E2 -9028.674} C_VEL
LIN {X 0,Y 439.363,Z 197.365,A -85,B 0,C 180,E1 -9032.031,E2 -9032.031} C_VEL
LIN {X 0,Y 439.39,Z 197.38,A -85,B 0,C 180,E1 -9035.341,E2 -9035.341} C_VEL
LIN {X 0,Y 439.379,Z 197.372,A -85,B 0,C 180,E1 -9038.595,E2 -9038.595} C_VEL
LIN {X 0,Y 439.383,Z 197.373,A -85,B 0,C 180,E1 -9041.257,E2 -9041.257} C_VEL
LIN {X 0,Y 439.394,Z 197.377,A -85,B 0,C 180,E1 -9044.73,E2 -9044.73} C_VEL
LIN {X 0,Y 439.391,Z 197.375,A -85,B 0,C 180,E1 -9047.796,E2 -9047.796} C_VEL
LIN {X 0,Y 439.384,Z 197.348,A -85,B 0,C 180,E1 -9050.224,E2 -9050.224} C_VEL
LIN {X 0,Y 439.369,Z 197.369,A -85,B 0,C 180,E1 -9053.713,E2 -9053.713} C_VEL
LIN {X 0,Y 439.374,Z 197.37,A -85,B 0,C 180,E1 -9057.055,E2 -9057.055} C_VEL
LIN {X 0,Y 439.42,Z 197.666,A -85,B 0,C 180,E1 -9057.449,E2 -9057.449} C_VEL
LIN {X 0,Y 444.015,Z 214.046,A -85,B 0,C 180,E1 -9060.269,E2 -9060.269} C_VEL
LIN {X 0,Y 446.348,Z 223.823,A -85,B 0,C 180,E1 -9061.854,E2 -9061.854} C_VEL
LIN {X 0,Y 445.787,Z 232.375,A -85,B 0,C 180,E1 -9063.048,E2 -9063.048} C_VEL
LIN {X 0,Y 444.907,Z 245.105,A -85,B 0,C 180,E1 -9064.775,E2 -9064.775} C_VEL
LIN {X 0,Y 448.821,Z 269.626,A -85,B 0,C 180,E1 -9065.45,E2 -9065.45} C_VEL
LIN {X 0,Y 446.562,Z 407.972,A -85,B 0,C 180,E1 -9067.839,E2 -9067.839} C_VEL
LIN {X 0,Y 445.905,Z 423.863,A -85,B 0,C 180,E1 -9068.292,E2 -9068.292} C_VEL
LIN {X 0,Y 445.129,Z 439.581,A -85,B 0,C 180,E1 -9068.95,E2 -9068.95} C_VEL
LIN {X 0,Y 444.214,Z 454.096,A -85,B 0,C 180,E1 -9069.752,E2 -9069.752} C_VEL
LIN {X 0,Y 443.273,Z 467.37,A -85,B 0,C 180,E1 -9070.673,E2 -9070.673} C_VEL
LIN {X 0,Y 442.263,Z 480.902,A -85,B 0,C 180,E1 -9071.829,E2 -9071.829} C_VEL
LIN {X 0,Y 441.405,Z 492.831,A -85,B 0,C 180,E1 -9073.06,E2 -9073.06} C_VEL
LIN {X 0,Y 440.509,Z 504.498,A -85,B 0,C 180,E1 -9074.501,E2 -9074.501} C_VEL
LIN {X 0,Y 439.884,Z 514.025,A -85,B 0,C 180,E1 -9075.899,E2 -9075.899} C_VEL
LIN {X 0,Y 439.199,Z 523.691,A -85,B 0,C 180,E1 -9077.593,E2 -9077.593} C_VEL
LIN {X 0,Y 438.871,Z 532.079,A -85,B 0,C 180,E1 -9079.388,E2 -9079.388} C_VEL
LIN {X 0,Y 438.516,Z 539.066,A -85,B 0,C 180,E1 -9081.243,E2 -9081.243} C_VEL
LIN {X 0,Y 438.399,Z 544.543,A -85,B 0,C 180,E1 -9083.095,E2 -9083.095} C_VEL
LIN {X 0,Y 438.343,Z 547.691,A -85,B 0,C 180,E1 -9084.48,E2 -9084.48} C_VEL
LIN {X 0,Y 438.296,Z 550.79,A -85,B 0,C 180,E1 -9086.323,E2 -9086.323} C_VEL
LIN {X 0,Y 438.316,Z 552.64,A -85,B 0,C 180,E1 -9088.163,E2 -9088.163} C_VEL
LIN {X 0,Y 438.306,Z 553.267,A -85,B 0,C 180,E1 -9090,E2 -9090} C_VEL
LIN {X 0,Y 438.316,Z 552.636,A -85,B 0,C 180,E1 -9091.838,E2 -9091.838} C_VEL
LIN {X 0,Y 438.297,Z 550.781,A -85,B 0,C 180,E1 -9093.678,E2 -9093.678} C_VEL
LIN {X 0,Y 438.363,Z 547.685,A -85,B 0,C 180,E1 -9095.52,E2 -9095.52} C_VEL
LIN {X 0,Y 438.478,Z 543.273,A -85,B 0,C 180,E1 -9097.367,E2 -9097.367} C_VEL
LIN {X 0,Y 438.572,Z 537.429,A -85,B 0,C 180,E1 -9099.221,E2 -9099.221} C_VEL
LIN {X 0,Y 438.976,Z 530.014,A -85,B 0,C 180,E1 -9101.077,E2 -9101.077} C_VEL
LIN {X 0,Y 439.351,Z 522.43,A -85,B 0,C 180,E1 -9102.637,E2 -9102.637} C_VEL
LIN {X 0,Y 439.982,Z 512.482,A -85,B 0,C 180,E1 -9104.335,E2 -9104.335} C_VEL
LIN {X 0,Y 440.647,Z 502.724,A -85,B 0,C 180,E1 -9105.732,E2 -9105.732} C_VEL
LIN {X 0,Y 441.535,Z 491.152,A -85,B 0,C 180,E1 -9107.123,E2 -9107.123} C_VEL
LIN {X 0,Y 442.354,Z 479.656,A -85,B 0,C 180,E1 -9108.287,E2 -9108.287} C_VEL
LIN {X 0,Y 443.405,Z 465.788,A -85,B 0,C 180,E1 -9109.442,E2 -9109.442} C_VEL
LIN {X 0,Y 444.325,Z 452.171,A -85,B 0,C 180,E1 -9110.364,E2 -9110.364} C_VEL
LIN {X 0,Y 445.234,Z 437.07,A -85,B 0,C 180,E1 -9111.167,E2 -9111.167} C_VEL
LIN {X 0,Y 445.998,Z 421.856,A -85,B 0,C 180,E1 -9111.77,E2 -9111.77} C_VEL
LIN {X 0,Y 446.558,Z 406.285,A -85,B 0,C 180,E1 -9112.192,E2 -9112.192} C_VEL
LIN {X 0,Y 448.795,Z 269.43,A -85,B 0,C 180,E1 -9114.549,E2 -9114.549} C_VEL
LIN {X 0,Y 444.858,Z 245.077,A -85,B 0,C 180,E1 -9115.224,E2 -9115.224} C_VEL
LIN {X 0,Y 446.429,Z 225.309,A -85,B 0,C 180,E1 -9117.932,E2 -9117.932} C_VEL
LIN {X 0,Y 445.896,Z 221.765,A -85,B 0,C 180,E1 -9118.476,E2 -9118.476} C_VEL
LIN {X 0,Y 442.151,Z 207.24,A -85,B 0,C 180,E1 -9120.87,E2 -9120.87} C_VEL
LIN {X 0,Y 439.412,Z 197.442,A -85,B 0,C 180,E1 -9122.611,E2 -9122.611} C_VEL
LIN {X 0,Y 439.39,Z 197.356,A -85,B 0,C 180,E1 -9125.34,E2 -9125.34} C_VEL
LIN {X 0,Y 439.368,Z 197.363,A -85,B 0,C 180,E1 -9128.596,E2 -9128.596} C_VEL
LIN {X 0,Y 439.387,Z 197.364,A -85,B 0,C 180,E1 -9131.257,E2 -9131.257} C_VEL
LIN {X 0,Y 439.398,Z 197.371,A -85,B 0,C 180,E1 -9134.729,E2 -9134.729} C_VEL
LIN {X 0,Y 439.394,Z 197.368,A -85,B 0,C 180,E1 -9137.796,E2 -9137.796} C_VEL
LIN {X 0,Y 439.435,Z 197.374,A -85,B 0,C 180,E1 -9140.228,E2 -9140.228} C_VEL
LIN {X 0,Y 439.371,Z 197.376,A -85,B 0,C 180,E1 -9143.713,E2 -9143.713} C_VEL
LIN {X 0,Y 439.37,Z 197.364,A -85,B 0,C 180,E1 -9147.054,E2 -9147.054} C_VEL
LIN {X 0,Y 439.38,Z 197.382,A -85,B 0,C 180,E1 -9150.274,E2 -9150.274} C_VEL
LIN {X 0,Y 439.425,Z 197.353,A -85,B 0,C 180,E1 -9153.396,E2 -9153.396} C_VEL
LIN {X 0,Y 439.382,Z 197.381,A -85,B 0,C 180,E1 -9156.429,E2 -9156.429} C_VEL
LIN {X 0,Y 439.385,Z 197.374,A -85,B 0,C 180,E1 -9159.397,E2 -9159.397} C_VEL
LIN {X 0,Y 439.428,Z 197.37,A -85,B 0,C 180,E1 -9162.31,E2 -9162.31} C_VEL
LIN {X 0,Y 439.445,Z 197.367,A -85,B 0,C 180,E1 -9165.174,E2 -9165.174} C_VEL
LIN {X 0,Y 439.481,Z 197.37,A -85,B 0,C 180,E1 -9168.001,E2 -9168.001} C_VEL
LIN {X 0,Y 439.545,Z 197.358,A -85,B 0,C 180,E1 -9171.726,E2 -9171.726} C_VEL
LIN {X 0,Y 439.618,Z 197.341,A -85,B 0,C 180,E1 -9174.496,E2 -9174.496} C_VEL
LIN {X 0,Y 439.631,Z 197.341,A -85,B 0,C 180,E1 -9178.168,E2 -9178.168} C_VEL
LIN {X 0,Y 439.759,Z 197.332,A -85,B 0,C 180,E1 -9180,E2 -9180} C_VEL
LIN {X 0,Y 439.638,Z 197.34,A -85,B 0,C 180,E1 -9182.749,E2 -9182.749} C_VEL
LIN {X 0,Y 439.615,Z 197.345,A -85,B 0,C 180,E1 -9186.425,E2 -9186.425} C_VEL
LIN {X 0,Y 439.498,Z 197.364,A -85,B 0,C 180,E1 -9189.202,E2 -9189.202} C_VEL
LIN {X 0,Y 439.464,Z 197.364,A -85,B 0,C 180,E1 -9192.938,E2 -9192.938} C_VEL
LIN {X 0,Y 439.445,Z 197.363,A -85,B 0,C 180,E1 -9196.349,E2 -9196.349} C_VEL
LIN {X 0,Y 439.401,Z 197.371,A -85,B 0,C 180,E1 -9199.627,E2 -9199.627} C_VEL
LIN {X 0,Y 439.363,Z 197.38,A -85,B 0,C 180,E1 -9202.576,E2 -9202.576} C_VEL
LIN {X 0,Y 439.404,Z 197.374,A -85,B 0,C 180,E1 -9205.585,E2 -9205.585} C_VEL
LIN {X 0,Y 439.416,Z 197.358,A -85,B 0,C 180,E1 -9208.674,E2 -9208.674} C_VEL
LIN {X 0,Y 439.369,Z 197.378,A -85,B 0,C 180,E1 -9212.031,E2 -9212.031} C_VEL
LIN {X 0,Y 439.396,Z 197.367,A -85,B 0,C 180,E1 -9215.341,E2 -9215.341} C_VEL
LIN {X 0,Y 439.38,Z 197.375,A -85,B 0,C 180,E1 -9218.596,E2 -9218.596} C_VEL
LIN {X 0,Y 439.388,Z 197.377,A -85,B 0,C 180,E1 -9221.257,E2 -9221.257} C_VEL
LIN {X 0,Y 439.401,Z 197.371,A -85,B 0,C 180,E1 -9224.73,E2 -9224.73} C_VEL
LIN {X 0,Y 439.396,Z 197.369,A -85,B 0,C 180,E1 -9227.796,E2 -9227.796} C_VEL
LIN {X 0,Y 439.427,Z 197.372,A -85,B 0,C 180,E1 -9230.228,E2 -9230.228} C_VEL
LIN {X 0,Y 439.375,Z 197.374,A -85,B 0,C 180,E1 -9233.713,E2 -9233.713} C_VEL
LIN {X 0,Y 439.374,Z 197.36,A -85,B 0,C 180,E1 -9237.054,E2 -9237.054} C_VEL
LIN {X 0,Y 439.42,Z 197.546,A -85,B 0,C 180,E1 -9239.24,E2 -9239.24} C_VEL
LIN {X 0,Y 443.052,Z 211.887,A -85,B 0,C 180,E1 -9242.099,E2 -9242.099} C_VEL
LIN {X 0,Y 444.944,Z 220.62,A -85,B 0,C 180,E1 -9243.751,E2 -9243.751} C_VEL
LIN {X 0,Y 443.896,Z 235.322,A -85,B 0,C 180,E1 -9246.188,E2 -9246.188} C_VEL
LIN {X 0,Y 443.39,Z 244.563,A -85,B 0,C 180,E1 -9247.662,E2 -9247.662} C_VEL
LIN {X 0,Y 448.156,Z 268.761,A -85,B 0,C 180,E1 -9248.34,E2 -9248.34} C_VEL
LIN {X 0,Y 446.908,Z 385.899,A -85,B 0,C 180,E1 -9250.149,E2 -9250.149} C_VEL
LIN {X 0,Y 446.806,Z 390.481,A -85,B 0,C 180,E1 -9250.259,E2 -9250.259} C_VEL
LIN {X 0,Y 446.037,Z 394.375,A -85,B 0,C 180,E1 -9250.328,E2 -9250.328} C_VEL
LIN {X 0,Y 440.201,Z 406.515,A -85,B 0,C 180,E1 -9250.479,E2 -9250.479} C_VEL
LIN {X 0,Y 439.46,Z 410.28,A -85,B 0,C 180,E1 -9250.616,E2 -9250.616} C_VEL
LIN {X 0,Y 438.624,Z 423.662,A -85,B 0,C 180,E1 -9251.309,E2 -9251.309} C_VEL
LIN {X 0,Y 437.888,Z 435.717,A -85,B 0,C 180,E1 -9252.124,E2 -9252.124} C_VEL
LIN {X 0,Y 436.794,Z 448.17,A -85,B 0,C 180,E1 -9253.165,E2 -9253.165} C_VEL
LIN {X 0,Y 435.86,Z 459.393,A -85,B 0,C 180,E1 -9254.331,E2 -9254.331} C_VEL
LIN {X 0,Y 434.92,Z 468.714,A -85,B 0,C 180,E1 -9255.495,E2 -9255.495} C_VEL
LIN {X 0,Y 434.101,Z 478.072,A -85,B 0,C 180,E1 -9256.9,E2 -9256.9} C_VEL
LIN {X 0,Y 433.304,Z 485.846,A -85,B 0,C 180,E1 -9258.302,E2 -9258.302} C_VEL
LIN {X 0,Y 432.708,Z 492.339,A -85,B 0,C 180,E1 -9259.708,E2 -9259.708} C_VEL
LIN {X 0,Y 432.113,Z 499.322,A -85,B 0,C 180,E1 -9261.583,E2 -9261.583} C_VEL
LIN {X 0,Y 431.778,Z 504.654,A -85,B 0,C 180,E1 -9263.457,E2 -9263.457} C_VEL
LIN {X 0,Y 431.422,Z 508.521,A -85,B 0,C 180,E1 -9265.328,E2 -9265.328} C_VEL
LIN {X 0,Y 431.39,Z 511.036,A -85,B 0,C 180,E1 -9267.198,E2 -9267.198} C_VEL
LIN {X 0,Y 431.237,Z 512.298,A -85,B 0,C 180,E1 -9269.066,E2 -9269.066} C_VEL
LIN {X 0,Y 431.236,Z 512.33,A -85,B 0,C 180,E1 -9270.933,E2 -9270.933} C_VEL
LIN {X 0,Y 431.387,Z 511.136,A -85,B 0,C 180,E1 -9272.801,E2 -9272.801} C_VEL
LIN {X 0,Y 431.41,Z 508.692,A -85,B 0,C 180,E1 -9274.672,E2 -9274.672} C_VEL
LIN {X 0,Y 431.778,Z 504.891,A -85,B 0,C 180,E1 -9276.542,E2 -9276.542} C_VEL
LIN {X 0,Y 432.08,Z 499.636,A -85,B 0,C 180,E1 -9278.417,E2 -9278.417} C_VEL
LIN {X 0,Y 432.64,Z 492.739,A -85,B 0,C 180,E1 -9280.293,E2 -9280.293} C_VEL
LIN {X 0,Y 433.375,Z 485.133,A -85,B 0,C 180,E1 -9281.932,E2 -9281.932} C_VEL
LIN {X 0,Y 434.205,Z 476.76,A -85,B 0,C 180,E1 -9283.408,E2 -9283.408} C_VEL
LIN {X 0,Y 435.04,Z 467.667,A -85,B 0,C 180,E1 -9284.74,E2 -9284.74} C_VEL
LIN {X 0,Y 436.078,Z 457.076,A -85,B 0,C 180,E1 -9286.021,E2 -9286.021} C_VEL
LIN {X 0,Y 436.963,Z 446.627,A -85,B 0,C 180,E1 -9287.069,E2 -9287.069} C_VEL
LIN {X 0,Y 438.02,Z 433.832,A -85,B 0,C 180,E1 -9288.111,E2 -9288.111} C_VEL
LIN {X 0,Y 438.836,Z 421.666,A -85,B 0,C 180,E1 -9288.898,E2 -9288.898} C_VEL
LIN {X 0,Y 439.477,Z 409.015,A -85,B 0,C 180,E1 -9289.537,E2 -9289.537} C_VEL
LIN {X 0,Y 440.067,Z 394.914,A -85,B 0,C 180,E1 -9290.051,E2 -9290.051} C_VEL
LIN {X 0,Y 440.376,Z 381.199,A -85,B 0,C 180,E1 -9290.371,E2 -9290.371} C_VEL
LIN {X 0,Y 441.59,Z 268.945,A -85,B 0,C 180,E1 -9292.117,E2 -9292.117} C_VEL
LIN {X 0,Y 436.635,Z 244.408,A -85,B 0,C 180,E1 -9292.839,E2 -9292.839} C_VEL
LIN {X 0,Y 438.156,Z 223.985,A -85,B 0,C 180,E1 -9296.229,E2 -9296.229} C_VEL
LIN {X 0,Y 437.654,Z 219.989,A -85,B 0,C 180,E1 -9296.963,E2 -9296.963} C_VEL
LIN {X 0,Y 434.5,Z 206.647,A -85,B 0,C 180,E1 -9299.574,E2 -9299.574} C_VEL
LIN {X 0,Y 432.373,Z 198.403,A -85,B 0,C 180,E1 -9301.284,E2 -9301.284} C_VEL
LIN {X 0,Y 432.339,Z 198.25,A -85,B 0,C 180,E1 -9304.676,E2 -9304.676} C_VEL
LIN {X 0,Y 432.343,Z 198.256,A -85,B 0,C 180,E1 -9308.148,E2 -9308.148} C_VEL
LIN {X 0,Y 432.33,Z 198.253,A -85,B 0,C 180,E1 -9311.601,E2 -9311.601} C_VEL
LIN {X 0,Y 432.334,Z 198.255,A -85,B 0,C 180,E1 -9314.346,E2 -9314.346} C_VEL
LIN {X 0,Y 432.316,Z 198.255,A -85,B 0,C 180,E1 -9317.015,E2 -9317.015} C_VEL
LIN {X 0,Y 432.329,Z 198.246,A -85,B 0,C 180,E1 -9319.82,E2 -9319.82} C_VEL
LIN {X 0,Y 432.311,Z 198.262,A -85,B 0,C 180,E1 -9323.022,E2 -9323.022} C_VEL
LIN {X 0,Y 432.355,Z 198.244,A -85,B 0,C 180,E1 -9325.996,E2 -9325.996} C_VEL
LIN {X 0,Y 432.39,Z 198.241,A -85,B 0,C 180,E1 -9329.743,E2 -9329.743} C_VEL
LIN {X 0,Y 432.394,Z 198.247,A -85,B 0,C 180,E1 -9333.372,E2 -9333.372} C_VEL
LIN {X 0,Y 432.365,Z 198.247,A -85,B 0,C 180,E1 -9336.023,E2 -9336.023} C_VEL
LIN {X 0,Y 432.343,Z 198.254,A -85,B 0,C 180,E1 -9339.046,E2 -9339.046} C_VEL
LIN {X 0,Y 432.372,Z 198.249,A -85,B 0,C 180,E1 -9342.011,E2 -9342.011} C_VEL
LIN {X 0,Y 432.39,Z 198.249,A -85,B 0,C 180,E1 -9344.926,E2 -9344.926} C_VEL
LIN {X 0,Y 432.452,Z 198.235,A -85,B 0,C 180,E1 -9347.803,E2 -9347.803} C_VEL
LIN {X 0,Y 432.485,Z 198.232,A -85,B 0,C 180,E1 -9351.59,E2 -9351.59} C_VEL
LIN {X 0,Y 432.591,Z 198.226,A -85,B 0,C 180,E1 -9354.406,E2 -9354.406} C_VEL
LIN {X 0,Y 432.598,Z 198.221,A -85,B 0,C 180,E1 -9358.138,E2 -9358.138} C_VEL
LIN {X 0,Y 432.726,Z 198.207,A -85,B 0,C 180,E1 -9360,E2 -9360} C_VEL
LIN {X 0,Y 432.598,Z 198.223,A -85,B 0,C 180,E1 -9362.793,E2 -9362.793} C_VEL
LIN {X 0,Y 432.565,Z 198.229,A -85,B 0,C 180,E1 -9366.53,E2 -9366.53} C_VEL
LIN {X 0,Y 432.435,Z 198.238,A -85,B 0,C 180,E1 -9369.353,E2 -9369.353} C_VEL
LIN {X 0,Y 432.423,Z 198.241,A -85,B 0,C 180,E1 -9372.803,E2 -9372.803} C_VEL
LIN {X 0,Y 432.405,Z 198.245,A -85,B 0,C 180,E1 -9376.479,E2 -9376.479} C_VEL
LIN {X 0,Y 432.332,Z 198.258,A -85,B 0,C 180,E1 -9379.961,E2 -9379.961} C_VEL
LIN {X 0,Y 432.312,Z 198.257,A -85,B 0,C 180,E1 -9382.964,E2 -9382.964} C_VEL
LIN {X 0,Y 432.357,Z 198.235,A -85,B 0,C 180,E1 -9386.033,E2 -9386.033} C_VEL
LIN {X 0,Y 432.336,Z 198.254,A -85,B 0,C 180,E1 -9389.188,E2 -9389.188} C_VEL
LIN {X 0,Y 432.316,Z 198.241,A -85,B 0,C 180,E1 -9392.443,E2 -9392.443} C_VEL
LIN {X 0,Y 432.339,Z 198.256,A -85,B 0,C 180,E1 -9395.632,E2 -9395.632} C_VEL
LIN {X 0,Y 432.349,Z 198.254,A -85,B 0,C 180,E1 -9399.343,E2 -9399.343} C_VEL
LIN {X 0,Y 432.327,Z 198.248,A -85,B 0,C 180,E1 -9401.798,E2 -9401.798} C_VEL
LIN {X 0,Y 432.328,Z 198.256,A -85,B 0,C 180,E1 -9404.348,E2 -9404.348} C_VEL
LIN {X 0,Y 432.315,Z 198.26,A -85,B 0,C 180,E1 -9407.016,E2 -9407.016} C_VEL
LIN {X 0,Y 432.328,Z 198.226,A -85,B 0,C 180,E1 -9409.821,E2 -9409.821} C_VEL
LIN {X 0,Y 432.302,Z 198.259,A -85,B 0,C 180,E1 -9413.023,E2 -9413.023} C_VEL
LIN {X 0,Y 432.328,Z 198.246,A -85,B 0,C 180,E1 -9416.002,E2 -9416.002} C_VEL
LIN {X 0,Y 432.361,Z 198.46,A -85,B 0,C 180,E1 -9416.991,E2 -9416.991} C_VEL
LIN {X 0,Y 437.36,Z 216.242,A -85,B 0,C 180,E1 -9420.124,E2 -9420.124} C_VEL
LIN {X 0,Y 439.67,Z 226.607,A -85,B 0,C 180,E1 -9421.821,E2 -9421.821} C_VEL
LIN {X 0,Y 438.214,Z 245.175,A -85,B 0,C 180,E1 -9424.393,E2 -9424.393} C_VEL
LIN {X 0,Y 442.285,Z 270.221,A -85,B 0,C 180,E1 -9425.099,E2 -9425.099} C_VEL
LIN {X 0,Y 439.948,Z 406.769,A -85,B 0,C 180,E1 -9427.488,E2 -9427.488} C_VEL
LIN {X 0,Y 439.362,Z 422.21,A -85,B 0,C 180,E1 -9427.921,E2 -9427.921} C_VEL
LIN {X 0,Y 438.569,Z 437.209,A -85,B 0,C 180,E1 -9428.53,E2 -9428.53} C_VEL
LIN {X 0,Y 437.637,Z 451.693,A -85,B 0,C 180,E1 -9429.312,E2 -9429.312} C_VEL
LIN {X 0,Y 436.654,Z 465.347,A -85,B 0,C 180,E1 -9430.246,E2 -9430.246} C_VEL
LIN {X 0,Y 435.707,Z 477.932,A -85,B 0,C 180,E1 -9431.302,E2 -9431.302} C_VEL
LIN {X 0,Y 434.73,Z 490.009,A -85,B 0,C 180,E1 -9432.519,E2 -9432.519} C_VEL
LIN {X 0,Y 433.94,Z 500.527,A -85,B 0,C 180,E1 -9433.778,E2 -9433.778} C_VEL
LIN {X 0,Y 433.114,Z 510.589,A -85,B 0,C 180,E1 -9435.193,E2 -9435.193} C_VEL
LIN {X 0,Y 432.418,Z 520.434,A -85,B 0,C 180,E1 -9436.848,E2 -9436.848} C_VEL
LIN {X 0,Y 431.945,Z 528.626,A -85,B 0,C 180,E1 -9438.504,E2 -9438.504} C_VEL
LIN {X 0,Y 431.547,Z 535.414,A -85,B 0,C 180,E1 -9440.155,E2 -9440.155} C_VEL
LIN {X 0,Y 431.367,Z 541.636,A -85,B 0,C 180,E1 -9442.04,E2 -9442.04} C_VEL
LIN {X 0,Y 431.263,Z 546.039,A -85,B 0,C 180,E1 -9443.759,E2 -9443.759} C_VEL
LIN {X 0,Y 431.23,Z 549.063,A -85,B 0,C 180,E1 -9445.326,E2 -9445.326} C_VEL
LIN {X 0,Y 431.278,Z 551.537,A -85,B 0,C 180,E1 -9447.198,E2 -9447.198} C_VEL
LIN {X 0,Y 431.216,Z 552.775,A -85,B 0,C 180,E1 -9449.067,E2 -9449.067} C_VEL
LIN {X 0,Y 431.216,Z 552.773,A -85,B 0,C 180,E1 -9450.934,E2 -9450.934} C_VEL
LIN {X 0,Y 431.278,Z 551.529,A -85,B 0,C 180,E1 -9452.802,E2 -9452.802} C_VEL
LIN {X 0,Y 431.235,Z 549.053,A -85,B 0,C 180,E1 -9454.674,E2 -9454.674} C_VEL
LIN {X 0,Y 431.337,Z 545.305,A -85,B 0,C 180,E1 -9456.549,E2 -9456.549} C_VEL
LIN {X 0,Y 431.4,Z 540.183,A -85,B 0,C 180,E1 -9458.431,E2 -9458.431} C_VEL
LIN {X 0,Y 431.659,Z 533.566,A -85,B 0,C 180,E1 -9460.317,E2 -9460.317} C_VEL
LIN {X 0,Y 432.107,Z 526.422,A -85,B 0,C 180,E1 -9461.969,E2 -9461.969} C_VEL
LIN {X 0,Y 432.587,Z 517.799,A -85,B 0,C 180,E1 -9463.626,E2 -9463.626} C_VEL
LIN {X 0,Y 433.26,Z 509.038,A -85,B 0,C 180,E1 -9465.043,E2 -9465.043} C_VEL
LIN {X 0,Y 434.054,Z 498.668,A -85,B 0,C 180,E1 -9466.46,E2 -9466.46} C_VEL
LIN {X 0,Y 434.979,Z 486.329,A -85,B 0,C 180,E1 -9467.878,E2 -9467.878} C_VEL
LIN {X 0,Y 435.963,Z 473.95,A -85,B 0,C 180,E1 -9469.053,E2 -9469.053} C_VEL
LIN {X 0,Y 437.011,Z 460.48,A -85,B 0,C 180,E1 -9470.106,E2 -9470.106} C_VEL
LIN {X 0,Y 438.089,Z 445.667,A -85,B 0,C 180,E1 -9471.033,E2 -9471.033} C_VEL
LIN {X 0,Y 438.889,Z 430.712,A -85,B 0,C 180,E1 -9471.757,E2 -9471.757} C_VEL
LIN {X 0,Y 439.623,Z 415.507,A -85,B 0,C 180,E1 -9472.289,E2 -9472.289} C_VEL
LIN {X 0,Y 440.087,Z 399.027,A -85,B 0,C 180,E1 -9472.66,E2 -9472.66} C_VEL
LIN {X 0,Y 442.192,Z 269.305,A -85,B 0,C 180,E1 -9474.917,E2 -9474.917} C_VEL
LIN {X 0,Y 438.176,Z 245.068,A -85,B 0,C 180,E1 -9475.609,E2 -9475.609} C_VEL
LIN {X 0,Y 439.682,Z 226.624,A -85,B 0,C 180,E1 -9478.181,E2 -9478.181} C_VEL
LIN {X 0,Y 436.894,Z 214.437,A -85,B 0,C 180,E1 -9480.178,E2 -9480.178} C_VEL
LIN {X 0,Y 432.349,Z 198.358,A -85,B 0,C 180,E1 -9483.028,E2 -9483.028} C_VEL
LIN {X 0,Y 432.336,Z 198.237,A -85,B 0,C 180,E1 -9485.818,E2 -9485.818} C_VEL
LIN {X 0,Y 432.321,Z 198.229,A -85,B 0,C 180,E1 -9489.346,E2 -9489.346} C_VEL
LIN {X 0,Y 432.332,Z 198.254,A -85,B 0,C 180,E1 -9491.797,E2 -9491.797} C_VEL
LIN {X 0,Y 432.332,Z 198.25,A -85,B 0,C 180,E1 -9494.347,E2 -9494.347} C_VEL
LIN {X 0,Y 432.318,Z 198.253,A -85,B 0,C 180,E1 -9497.016,E2 -9497.016} C_VEL
LIN {X 0,Y 432.339,Z 198.255,A -85,B 0,C 180,E1 -9499.82,E2 -9499.82} C_VEL
LIN {X 0,Y 432.304,Z 198.254,A -85,B 0,C 180,E1 -9503.022,E2 -9503.022} C_VEL
LIN {X 0,Y 432.357,Z 198.253,A -85,B 0,C 180,E1 -9505.997,E2 -9505.997} C_VEL
LIN {X 0,Y 432.345,Z 198.251,A -85,B 0,C 180,E1 -9509.49,E2 -9509.49} C_VEL
LIN {X 0,Y 432.388,Z 198.23,A -85,B 0,C 180,E1 -9512.928,E2 -9512.928} C_VEL
LIN {X 0,Y 432.365,Z 198.251,A -85,B 0,C 180,E1 -9516.023,E2 -9516.023} C_VEL
LIN {X 0,Y 432.347,Z 198.25,A -85,B 0,C 180,E1 -9519.046,E2 -9519.046} C_VEL
LIN {X 0,Y 432.375,Z 198.249,A -85,B 0,C 180,E1 -9522.011,E2 -9522.011} C_VEL
LIN {X 0,Y 432.392,Z 198.245,A -85,B 0,C 180,E1 -9524.927,E2 -9524.927} C_VEL
LIN {X 0,Y 432.456,Z 198.242,A -85,B 0,C 180,E1 -9527.804,E2 -9527.804} C_VEL
LIN {X 0,Y 432.489,Z 198.235,A -85,B 0,C 180,E1 -9531.59,E2 -9531.59} C_VEL
LIN {X 0,Y 432.594,Z 198.217,A -85,B 0,C 180,E1 -9534.406,E2 -9534.406} C_VEL
LIN {X 0,Y 432.601,Z 198.216,A -85,B 0,C 180,E1 -9538.138,E2 -9538.138} C_VEL
LIN {X 0,Y 432.729,Z 198.207,A -85,B 0,C 180,E1 -9540,E2 -9540} C_VEL
LIN {X 0,Y 432.59,Z 198.218,A -85,B 0,C 180,E1 -9542.794,E2 -9542.794} C_VEL
LIN {X 0,Y 432.57,Z 198.223,A -85,B 0,C 180,E1 -9546.531,E2 -9546.531} C_VEL
LIN {X 0,Y 432.44,Z 198.245,A -85,B 0,C 180,E1 -9549.353,E2 -9549.353} C_VEL
LIN {X 0,Y 432.429,Z 198.239,A -85,B 0,C 180,E1 -9552.804,E2 -9552.804} C_VEL
LIN {X 0,Y 432.411,Z 198.239,A -85,B 0,C 180,E1 -9556.479,E2 -9556.479} C_VEL
LIN {X 0,Y 432.337,Z 198.249,A -85,B 0,C 180,E1 -9559.961,E2 -9559.961} C_VEL
LIN {X 0,Y 432.317,Z 198.258,A -85,B 0,C 180,E1 -9562.965,E2 -9562.965} C_VEL
LIN {X 0,Y 432.363,Z 198.25,A -85,B 0,C 180,E1 -9566.033,E2 -9566.033} C_VEL
LIN {X 0,Y 432.341,Z 198.239,A -85,B 0,C 180,E1 -9569.188,E2 -9569.188} C_VEL
LIN {X 0,Y 432.322,Z 198.259,A -85,B 0,C 180,E1 -9572.443,E2 -9572.443} C_VEL
LIN {X 0,Y 432.345,Z 198.247,A -85,B 0,C 180,E1 -9575.632,E2 -9575.632} C_VEL
LIN {X 0,Y 432.342,Z 198.25,A -85,B 0,C 180,E1 -9578.715,E2 -9578.715} C_VEL
LIN {X 0,Y 432.333,Z 198.255,A -85,B 0,C 180,E1 -9581.797,E2 -9581.797} C_VEL
LIN {X 0,Y 432.334,Z 198.248,A -85,B 0,C 180,E1 -9584.348,E2 -9584.348} C_VEL
LIN {X 0,Y 432.323,Z 198.252,A -85,B 0,C 180,E1 -9587.016,E2 -9587.016} C_VEL
LIN {X 0,Y 432.334,Z 198.258,A -85,B 0,C 180,E1 -9589.821,E2 -9589.821} C_VEL
LIN {X 0,Y 432.311,Z 198.255,A -85,B 0,C 180,E1 -9593.023,E2 -9593.023} C_VEL
LIN {X 0,Y 432.361,Z 198.237,A -85,B 0,C 180,E1 -9595.997,E2 -9595.997} C_VEL
LIN {X 0,Y 432.37,Z 198.406,A -85,B 0,C 180,E1 -9598.819,E2 -9598.819} C_VEL
LIN {X 0,Y 436.195,Z 213.475,A -85,B 0,C 180,E1 -9601.883,E2 -9601.883} C_VEL
LIN {X 0,Y 438.095,Z 221.935,A -85,B 0,C 180,E1 -9603.516,E2 -9603.516} C_VEL
LIN {X 0,Y 437.343,Z 233.997,A -85,B 0,C 180,E1 -9605.556,E2 -9605.556} C_VEL
LIN {X 0,Y 436.614,Z 244.358,A -85,B 0,C 180,E1 -9607.251,E2 -9607.251} C_VEL
LIN {X 0,Y 440.032,Z 261.11,A -85,B 0,C 180,E1 -9607.76,E2 -9607.76} C_VEL
LIN {X 0,Y 441.653,Z 270.162,A -85,B 0,C 180,E1 -9608.002,E2 -9608.002} C_VEL
LIN {X 0,Y 440.325,Z 385.693,A -85,B 0,C 180,E1 -9609.809,E2 -9609.809} C_VEL
LIN {X 0,Y 439.848,Z 400.27,A -85,B 0,C 180,E1 -9610.212,E2 -9610.212} C_VEL
LIN {X 0,Y 439.46,Z 410.28,A -85,B 0,C 180,E1 -9610.616,E2 -9610.616} C_VEL
LIN {X 0,Y 438.644,Z 415.847,A -85,B 0,C 180,E1 -9610.852,E2 -9610.852} C_VEL
LIN {X 0,Y 435.449,Z 424.821,A -85,B 0,C 180,E1 -9611.216,E2 -9611.216} C_VEL
LIN {X 0,Y 432.07,Z 433.515,A -85,B 0,C 180,E1 -9611.662,E2 -9611.662} C_VEL
LIN {X 0,Y 430.977,Z 438.641,A -85,B 0,C 180,E1 -9612.023,E2 -9612.023} C_VEL
LIN {X 0,Y 429.798,Z 451.041,A -85,B 0,C 180,E1 -9613.127,E2 -9613.127} C_VEL
LIN {X 0,Y 428.826,Z 461.798,A -85,B 0,C 180,E1 -9614.311,E2 -9614.311} C_VEL
LIN {X 0,Y 427.766,Z 472.418,A -85,B 0,C 180,E1 -9615.733,E2 -9615.733} C_VEL
LIN {X 0,Y 426.934,Z 481.193,A -85,B 0,C 180,E1 -9617.16,E2 -9617.16} C_VEL
LIN {X 0,Y 426.037,Z 489.6,A -85,B 0,C 180,E1 -9618.823,E2 -9618.823} C_VEL
LIN {X 0,Y 425.354,Z 496.406,A -85,B 0,C 180,E1 -9620.489,E2 -9620.489} C_VEL
LIN {X 0,Y 424.845,Z 502.531,A -85,B 0,C 180,E1 -9622.395,E2 -9622.395} C_VEL
LIN {X 0,Y 424.538,Z 507.102,A -85,B 0,C 180,E1 -9624.299,E2 -9624.299} C_VEL
LIN {X 0,Y 424.394,Z 510.273,A -85,B 0,C 180,E1 -9626.202,E2 -9626.202} C_VEL
LIN {X 0,Y 424.22,Z 512.155,A -85,B 0,C 180,E1 -9628.101,E2 -9628.101} C_VEL
LIN {X 0,Y 424.139,Z 512.798,A -85,B 0,C 180,E1 -9630,E2 -9630} C_VEL
LIN {X 0,Y 424.208,Z 512.22,A -85,B 0,C 180,E1 -9631.898,E2 -9631.898} C_VEL
LIN {X 0,Y 424.369,Z 510.408,A -85,B 0,C 180,E1 -9633.798,E2 -9633.798} C_VEL
LIN {X 0,Y 424.536,Z 507.305,A -85,B 0,C 180,E1 -9635.7,E2 -9635.7} C_VEL
LIN {X 0,Y 424.83,Z 502.802,A -85,B 0,C 180,E1 -9637.605,E2 -9637.605} C_VEL
LIN {X 0,Y 425.332,Z 496.758,A -85,B 0,C 180,E1 -9639.51,E2 -9639.51} C_VEL
LIN {X 0,Y 426.016,Z 490.035,A -85,B 0,C 180,E1 -9641.176,E2 -9641.176} C_VEL
LIN {X 0,Y 426.858,Z 481.717,A -85,B 0,C 180,E1 -9642.842,E2 -9642.842} C_VEL
LIN {X 0,Y 427.692,Z 473.05,A -85,B 0,C 180,E1 -9644.269,E2 -9644.269} C_VEL
LIN {X 0,Y 428.719,Z 462.553,A -85,B 0,C 180,E1 -9645.693,E2 -9645.693} C_VEL
LIN {X 0,Y 429.719,Z 451.944,A -85,B 0,C 180,E1 -9646.875,E2 -9646.875} C_VEL
LIN {X 0,Y 430.864,Z 440.344,A -85,B 0,C 180,E1 -9647.931,E2 -9647.931} C_VEL
LIN {X 0,Y 431.736,Z 427.563,A -85,B 0,C 180,E1 -9648.876,E2 -9648.876} C_VEL
LIN {X 0,Y 432.577,Z 415.03,A -85,B 0,C 180,E1 -9649.594,E2 -9649.594} C_VEL
LIN {X 0,Y 433.239,Z 401.109,A -85,B 0,C 180,E1 -9650.195,E2 -9650.195} C_VEL
LIN {X 0,Y 433.723,Z 387,A -85,B 0,C 180,E1 -9650.605,E2 -9650.605} C_VEL
LIN {X 0,Y 435.103,Z 270.085,A -85,B 0,C 180,E1 -9652.471,E2 -9652.471} C_VEL
LIN {X 0,Y 429.91,Z 244.493,A -85,B 0,C 180,E1 -9653.237,E2 -9653.237} C_VEL
LIN {X 0,Y 431.347,Z 225.993,A -85,B 0,C 180,E1 -9656.346,E2 -9656.346} C_VEL
LIN {X 0,Y 431.093,Z 222.903,A -85,B 0,C 180,E1 -9656.913,E2 -9656.913} C_VEL
LIN {X 0,Y 428.034,Z 209.749,A -85,B 0,C 180,E1 -9659.515,E2 -9659.515} C_VEL
LIN {X 0,Y 425.303,Z 199.226,A -85,B 0,C 180,E1 -9661.749,E2 -9661.749} C_VEL
LIN {X 0,Y 425.299,Z 199.134,A -85,B 0,C 180,E1 -9665.335,E2 -9665.335} C_VEL
LIN {X 0,Y 425.307,Z 199.128,A -85,B 0,C 180,E1 -9668.897,E2 -9668.897} C_VEL
LIN {X 0,Y 425.287,Z 199.127,A -85,B 0,C 180,E1 -9671.957,E2 -9671.957} C_VEL
LIN {X 0,Y 425.282,Z 199.129,A -85,B 0,C 180,E1 -9675.282,E2 -9675.282} C_VEL
LIN {X 0,Y 425.27,Z 199.136,A -85,B 0,C 180,E1 -9678.621,E2 -9678.621} C_VEL
LIN {X 0,Y 425.296,Z 199.124,A -85,B 0,C 180,E1 -9681.101,E2 -9681.101} C_VEL
LIN {X 0,Y 425.296,Z 199.123,A -85,B 0,C 180,E1 -9684.664,E2 -9684.664} C_VEL
LIN {X 0,Y 425.261,Z 199.136,A -85,B 0,C 180,E1 -9688.072,E2 -9688.072} C_VEL
LIN {X 0,Y 425.332,Z 199.11,A -85,B 0,C 180,E1 -9691.368,E2 -9691.368} C_VEL
LIN {X 0,Y 425.29,Z 199.133,A -85,B 0,C 180,E1 -9694.554,E2 -9694.554} C_VEL
LIN {X 0,Y 425.282,Z 199.133,A -85,B 0,C 180,E1 -9697.661,E2 -9697.661} C_VEL
LIN {X 0,Y 425.355,Z 199.122,A -85,B 0,C 180,E1 -9700.704,E2 -9700.704} C_VEL
LIN {X 0,Y 425.382,Z 199.115,A -85,B 0,C 180,E1 -9703.688,E2 -9703.688} C_VEL
LIN {X 0,Y 425.387,Z 199.118,A -85,B 0,C 180,E1 -9707.095,E2 -9707.095} C_VEL
LIN {X 0,Y 425.394,Z 199.123,A -85,B 0,C 180,E1 -9710.49,E2 -9710.49} C_VEL
LIN {X 0,Y 425.524,Z 199.101,A -85,B 0,C 180,E1 -9713.361,E2 -9713.361} C_VEL
LIN {X 0,Y 425.363,Z 199.122,A -85,B 0,C 180,E1 -9715.261,E2 -9715.261} C_VEL
LIN {X 0,Y 425.568,Z 199.096,A -85,B 0,C 180,E1 -9718.107,E2 -9718.107} C_VEL
LIN {X 0,Y 425.696,Z 199.083,A -85,B 0,C 180,E1 -9720,E2 -9720} C_VEL
LIN {X 0,Y 425.55,Z 199.101,A -85,B 0,C 180,E1 -9722.84,E2 -9722.84} C_VEL
LIN {X 0,Y 425.524,Z 199.105,A -85,B 0,C 180,E1 -9726.639,E2 -9726.639} C_VEL
LIN {X 0,Y 425.394,Z 199.116,A -85,B 0,C 180,E1 -9729.509,E2 -9729.509} C_VEL
LIN {X 0,Y 425.386,Z 199.117,A -85,B 0,C 180,E1 -9732.904,E2 -9732.904} C_VEL
LIN {X 0,Y 425.354,Z 199.122,A -85,B 0,C 180,E1 -9736.605,E2 -9736.605} C_VEL
LIN {X 0,Y 425.321,Z 199.13,A -85,B 0,C 180,E1 -9739.636,E2 -9739.636} C_VEL
LIN {X 0,Y 425.3,Z 199.132,A -85,B 0,C 180,E1 -9743.365,E2 -9743.365} C_VEL
LIN {X 0,Y 425.341,Z 199.107,A -85,B 0,C 180,E1 -9746.845,E2 -9746.845} C_VEL
LIN {X 0,Y 425.284,Z 199.138,A -85,B 0,C 180,E1 -9749.72,E2 -9749.72} C_VEL
LIN {X 0,Y 425.275,Z 199.119,A -85,B 0,C 180,E1 -9753.048,E2 -9753.048} C_VEL
LIN {X 0,Y 425.277,Z 199.132,A -85,B 0,C 180,E1 -9755.929,E2 -9755.929} C_VEL
LIN {X 0,Y 425.295,Z 199.129,A -85,B 0,C 180,E1 -9759.044,E2 -9759.044} C_VEL
LIN {X 0,Y 425.269,Z 199.129,A -85,B 0,C 180,E1 -9762.654,E2 -9762.654} C_VEL
LIN {X 0,Y 425.256,Z 199.133,A -85,B 0,C 180,E1 -9766.045,E2 -9766.045} C_VEL
LIN {X 0,Y 425.269,Z 199.122,A -85,B 0,C 180,E1 -9768.622,E2 -9768.622} C_VEL
LIN {X 0,Y 425.288,Z 199.109,A -85,B 0,C 180,E1 -9771.101,E2 -9771.101} C_VEL
LIN {X 0,Y 425.291,Z 199.11,A -85,B 0,C 180,E1 -9774.664,E2 -9774.664} C_VEL
LIN {X 0,Y 425.299,Z 199.33,A -85,B 0,C 180,E1 -9776.53,E2 -9776.53} C_VEL
LIN {X 0,Y 429.657,Z 214.626,A -85,B 0,C 180,E1 -9779.307,E2 -9779.307} C_VEL
LIN {X 0,Y 432.879,Z 227.942,A -85,B 0,C 180,E1 -9781.564,E2 -9781.564} C_VEL
LIN {X 0,Y 431.536,Z 245.254,A -85,B 0,C 180,E1 -9783.998,E2 -9783.998} C_VEL
LIN {X 0,Y 435.779,Z 270.912,A -85,B 0,C 180,E1 -9784.74,E2 -9784.74} C_VEL
LIN {X 0,Y 433.322,Z 407.305,A -85,B 0,C 180,E1 -9787.162,E2 -9787.162} C_VEL
LIN {X 0,Y 432.681,Z 422.803,A -85,B 0,C 180,E1 -9787.612,E2 -9787.612} C_VEL
LIN {X 0,Y 431.855,Z 437.906,A -85,B 0,C 180,E1 -9788.246,E2 -9788.246} C_VEL
LIN {X 0,Y 430.83,Z 453.038,A -85,B 0,C 180,E1 -9789.094,E2 -9789.094} C_VEL
LIN {X 0,Y 429.793,Z 466.411,A -85,B 0,C 180,E1 -9790.042,E2 -9790.042} C_VEL
LIN {X 0,Y 428.823,Z 478.783,A -85,B 0,C 180,E1 -9791.115,E2 -9791.115} C_VEL
LIN {X 0,Y 427.792,Z 490.556,A -85,B 0,C 180,E1 -9792.336,E2 -9792.336} C_VEL
LIN {X 0,Y 426.883,Z 501.943,A -85,B 0,C 180,E1 -9793.748,E2 -9793.748} C_VEL
LIN {X 0,Y 426.048,Z 511.724,A -85,B 0,C 180,E1 -9795.186,E2 -9795.186} C_VEL
LIN {X 0,Y 425.307,Z 521.504,A -85,B 0,C 180,E1 -9796.902,E2 -9796.902} C_VEL
LIN {X 0,Y 424.848,Z 529.303,A -85,B 0,C 180,E1 -9798.551,E2 -9798.551} C_VEL
LIN {X 0,Y 424.412,Z 536.73,A -85,B 0,C 180,E1 -9800.469,E2 -9800.469} C_VEL
LIN {X 0,Y 424.238,Z 542.581,A -85,B 0,C 180,E1 -9802.385,E2 -9802.385} C_VEL
LIN {X 0,Y 424.158,Z 547.01,A -85,B 0,C 180,E1 -9804.295,E2 -9804.295} C_VEL
LIN {X 0,Y 424.106,Z 550.118,A -85,B 0,C 180,E1 -9806.2,E2 -9806.2} C_VEL
LIN {X 0,Y 424.162,Z 551.974,A -85,B 0,C 180,E1 -9808.101,E2 -9808.101} C_VEL
LIN {X 0,Y 424.131,Z 552.602,A -85,B 0,C 180,E1 -9810,E2 -9810} C_VEL
LIN {X 0,Y 424.163,Z 551.97,A -85,B 0,C 180,E1 -9811.899,E2 -9811.899} C_VEL
LIN {X 0,Y 424.107,Z 550.108,A -85,B 0,C 180,E1 -9813.801,E2 -9813.801} C_VEL
LIN {X 0,Y 424.187,Z 547.002,A -85,B 0,C 180,E1 -9815.705,E2 -9815.705} C_VEL
LIN {X 0,Y 424.292,Z 542.575,A -85,B 0,C 180,E1 -9817.615,E2 -9817.615} C_VEL
LIN {X 0,Y 424.413,Z 536.714,A -85,B 0,C 180,E1 -9819.532,E2 -9819.532} C_VEL
LIN {X 0,Y 424.85,Z 529.277,A -85,B 0,C 180,E1 -9821.45,E2 -9821.45} C_VEL
LIN {X 0,Y 425.297,Z 521.993,A -85,B 0,C 180,E1 -9823,E2 -9823} C_VEL
LIN {X 0,Y 425.932,Z 513.215,A -85,B 0,C 180,E1 -9824.574,E2 -9824.574} C_VEL
LIN {X 0,Y 426.671,Z 503.663,A -85,B 0,C 180,E1 -9826.016,E2 -9826.016} C_VEL
LIN {X 0,Y 427.677,Z 492.06,A -85,B 0,C 180,E1 -9827.489,E2 -9827.489} C_VEL
LIN {X 0,Y 428.634,Z 479.965,A -85,B 0,C 180,E1 -9828.771,E2 -9828.771} C_VEL
LIN {X 0,Y 429.8,Z 466.336,A -85,B 0,C 180,E1 -9829.959,E2 -9829.959} C_VEL
LIN {X 0,Y 430.805,Z 452.939,A -85,B 0,C 180,E1 -9830.908,E2 -9830.908} C_VEL
LIN {X 0,Y 431.819,Z 437.826,A -85,B 0,C 180,E1 -9831.755,E2 -9831.755} C_VEL
LIN {X 0,Y 432.672,Z 422.14,A -85,B 0,C 180,E1 -9832.407,E2 -9832.407} C_VEL
LIN {X 0,Y 433.299,Z 406.998,A -85,B 0,C 180,E1 -9832.84,E2 -9832.84} C_VEL
LIN {X 0,Y 435.728,Z 271.718,A -85,B 0,C 180,E1 -9835.241,E2 -9835.241} C_VEL
LIN {X 0,Y 434.511,Z 263.096,A -85,B 0,C 180,E1 -9835.471,E2 -9835.471} C_VEL
LIN {X 0,Y 431.503,Z 244.993,A -85,B 0,C 180,E1 -9836.013,E2 -9836.013} C_VEL
LIN {X 0,Y 432.908,Z 227.949,A -85,B 0,C 180,E1 -9838.437,E2 -9838.437} C_VEL
LIN {X 0,Y 429.655,Z 214.582,A -85,B 0,C 180,E1 -9840.694,E2 -9840.694} C_VEL
LIN {X 0,Y 425.297,Z 199.231,A -85,B 0,C 180,E1 -9843.489,E2 -9843.489} C_VEL
LIN {X 0,Y 425.263,Z 199.128,A -85,B 0,C 180,E1 -9846.509,E2 -9846.509} C_VEL
LIN {X 0,Y 425.275,Z 199.108,A -85,B 0,C 180,E1 -9849.04,E2 -9849.04} C_VEL
LIN {X 0,Y 425.289,Z 199.131,A -85,B 0,C 180,E1 -9851.958,E2 -9851.958} C_VEL
LIN {X 0,Y 425.283,Z 199.134,A -85,B 0,C 180,E1 -9855.283,E2 -9855.283} C_VEL
LIN {X 0,Y 425.273,Z 199.129,A -85,B 0,C 180,E1 -9858.621,E2 -9858.621} C_VEL
LIN {X 0,Y 425.31,Z 199.127,A -85,B 0,C 180,E1 -9861.103,E2 -9861.103} C_VEL
LIN {X 0,Y 425.297,Z 199.137,A -85,B 0,C 180,E1 -9864.664,E2 -9864.664} C_VEL
LIN {X 0,Y 425.262,Z 199.122,A -85,B 0,C 180,E1 -9868.073,E2 -9868.073} C_VEL
LIN {X 0,Y 425.328,Z 199.125,A -85,B 0,C 180,E1 -9871.368,E2 -9871.368} C_VEL
LIN {X 0,Y 425.351,Z 199.104,A -85,B 0,C 180,E1 -9873.505,E2 -9873.505} C_VEL
LIN {X 0,Y 425.302,Z 199.132,A -85,B 0,C 180,E1 -9876.635,E2 -9876.635} C_VEL
LIN {X 0,Y 425.326,Z 199.13,A -85,B 0,C 180,E1 -9880.364,E2 -9880.364} C_VEL
LIN {X 0,Y 425.386,Z 199.121,A -85,B 0,C 180,E1 -9883.688,E2 -9883.688} C_VEL
LIN {X 0,Y 425.409,Z 199.117,A -85,B 0,C 180,E1 -9887.598,E2 -9887.598} C_VEL
LIN {X 0,Y 425.44,Z 199.112,A -85,B 0,C 180,E1 -9891.45,E2 -9891.45} C_VEL
LIN {X 0,Y 425.551,Z 199.094,A -85,B 0,C 180,E1 -9894.313,E2 -9894.313} C_VEL
LIN {X 0,Y 425.571,Z 199.092,A -85,B 0,C 180,E1 -9898.107,E2 -9898.107} C_VEL
LIN {X 0,Y 425.699,Z 199.083,A -85,B 0,C 180,E1 -9900,E2 -9900} C_VEL
LIN {X 0,Y 425.544,Z 199.096,A -85,B 0,C 180,E1 -9902.84,E2 -9902.84} C_VEL
LIN {X 0,Y 425.529,Z 199.1,A -85,B 0,C 180,E1 -9906.639,E2 -9906.639} C_VEL
LIN {X 0,Y 425.399,Z 199.123,A -85,B 0,C 180,E1 -9909.51,E2 -9909.51} C_VEL
LIN {X 0,Y 425.391,Z 199.117,A -85,B 0,C 180,E1 -9912.904,E2 -9912.904} C_VEL
LIN {X 0,Y 425.36,Z 199.118,A -85,B 0,C 180,E1 -9916.605,E2 -9916.605} C_VEL
LIN {X 0,Y 425.327,Z 199.123,A -85,B 0,C 180,E1 -9919.636,E2 -9919.636} C_VEL
LIN {X 0,Y 425.305,Z 199.128,A -85,B 0,C 180,E1 -9923.365,E2 -9923.365} C_VEL
LIN {X 0,Y 425.346,Z 199.122,A -85,B 0,C 180,E1 -9926.844,E2 -9926.844} C_VEL
LIN {X 0,Y 425.29,Z 199.123,A -85,B 0,C 180,E1 -9929.72,E2 -9929.72} C_VEL
LIN {X 0,Y 425.281,Z 199.13,A -85,B 0,C 180,E1 -9933.048,E2 -9933.048} C_VEL
LIN {X 0,Y 425.284,Z 199.126,A -85,B 0,C 180,E1 -9935.929,E2 -9935.929} C_VEL
LIN {X 0,Y 425.283,Z 199.124,A -85,B 0,C 180,E1 -9939.041,E2 -9939.041} C_VEL
LIN {X 0,Y 425.289,Z 199.133,A -85,B 0,C 180,E1 -9941.958,E2 -9941.958} C_VEL
LIN {X 0,Y 425.285,Z 199.133,A -85,B 0,C 180,E1 -9945.283,E2 -9945.283} C_VEL
LIN {X 0,Y 425.275,Z 199.133,A -85,B 0,C 180,E1 -9948.622,E2 -9948.622} C_VEL
LIN {X 0,Y 425.31,Z 199.126,A -85,B 0,C 180,E1 -9951.103,E2 -9951.103} C_VEL
LIN {X 0,Y 425.301,Z 199.135,A -85,B 0,C 180,E1 -9954.664,E2 -9954.664} C_VEL
LIN {X 0,Y 425.317,Z 199.171,A -85,B 0,C 180,E1 -9958.321,E2 -9958.321} C_VEL
LIN {X 0,Y 426.143,Z 202.301,A -85,B 0,C 180,E1 -9959.047,E2 -9959.047} C_VEL
LIN {X 0,Y 429.358,Z 215.073,A -85,B 0,C 180,E1 -9961.661,E2 -9961.661} C_VEL
LIN {X 0,Y 431.285,Z 223.662,A -85,B 0,C 180,E1 -9963.348,E2 -9963.348} C_VEL
LIN {X 0,Y 430.727,Z 232.671,A -85,B 0,C 180,E1 -9964.898,E2 -9964.898} C_VEL
LIN {X 0,Y 429.884,Z 244.494,A -85,B 0,C 180,E1 -9966.859,E2 -9966.859} C_VEL
LIN {X 0,Y 435.152,Z 270.687,A -85,B 0,C 180,E1 -9967.638,E2 -9967.638} C_VEL
LIN {X 0,Y 433.708,Z 386.851,A -85,B 0,C 180,E1 -9969.487,E2 -9969.487} C_VEL
LIN {X 0,Y 433.232,Z 401.02,A -85,B 0,C 180,E1 -9969.897,E2 -9969.897} C_VEL
LIN {X 0,Y 432.679,Z 413.599,A -85,B 0,C 180,E1 -9970.428,E2 -9970.428} C_VEL
LIN {X 0,Y 431.869,Z 426.169,A -85,B 0,C 180,E1 -9971.129,E2 -9971.129} C_VEL
LIN {X 0,Y 430.977,Z 438.641,A -85,B 0,C 180,E1 -9972.023,E2 -9972.023} C_VEL
LIN {X 0,Y 429.884,Z 443.736,A -85,B 0,C 180,E1 -9972.415,E2 -9972.415} C_VEL
LIN {X 0,Y 426.415,Z 451.739,A -85,B 0,C 180,E1 -9973.041,E2 -9973.041} C_VEL
LIN {X 0,Y 422.94,Z 459.402,A -85,B 0,C 180,E1 -9973.743,E2 -9973.743} C_VEL
LIN {X 0,Y 421.84,Z 463.782,A -85,B 0,C 180,E1 -9974.248,E2 -9974.248} C_VEL
LIN {X 0,Y 420.799,Z 473.67,A -85,B 0,C 180,E1 -9975.626,E2 -9975.626} C_VEL
LIN {X 0,Y 419.861,Z 482.884,A -85,B 0,C 180,E1 -9977.186,E2 -9977.186} C_VEL
LIN {X 0,Y 418.965,Z 491.044,A -85,B 0,C 180,E1 -9978.877,E2 -9978.877} C_VEL
LIN {X 0,Y 418.349,Z 496.759,A -85,B 0,C 180,E1 -9980.329,E2 -9980.329} C_VEL
LIN {X 0,Y 417.824,Z 502.876,A -85,B 0,C 180,E1 -9982.266,E2 -9982.266} C_VEL
LIN {X 0,Y 417.501,Z 507.442,A -85,B 0,C 180,E1 -9984.203,E2 -9984.203} C_VEL
LIN {X 0,Y 417.301,Z 510.611,A -85,B 0,C 180,E1 -9986.137,E2 -9986.137} C_VEL
LIN {X 0,Y 417.146,Z 512.489,A -85,B 0,C 180,E1 -9988.069,E2 -9988.069} C_VEL
LIN {X 0,Y 417.056,Z 513.131,A -85,B 0,C 180,E1 -9990,E2 -9990} C_VEL
LIN {X 0,Y 417.135,Z 512.553,A -85,B 0,C 180,E1 -9991.931,E2 -9991.931} C_VEL
LIN {X 0,Y 417.277,Z 510.744,A -85,B 0,C 180,E1 -9993.863,E2 -9993.863} C_VEL
LIN {X 0,Y 417.496,Z 507.642,A -85,B 0,C 180,E1 -9995.796,E2 -9995.796} C_VEL
LIN {X 0,Y 417.783,Z 503.146,A -85,B 0,C 180,E1 -9997.734,E2 -9997.734} C_VEL
LIN {X 0,Y 418.324,Z 497.108,A -85,B 0,C 180,E1 -9999.671,E2 -9999.671} C_VEL
LIN {X 0,Y 419.019,Z 490.395,A -85,B 0,C 180,E1 -10001.366,E2 -10001.366} C_VEL
LIN {X 0,Y 419.94,Z 482.086,A -85,B 0,C 180,E1 -10003.057,E2 -10003.057} C_VEL
LIN {X 0,Y 420.797,Z 473.434,A -85,B 0,C 180,E1 -10004.508,E2 -10004.508} C_VEL
LIN {X 0,Y 421.908,Z 462.954,A -85,B 0,C 180,E1 -10005.953,E2 -10005.953} C_VEL
LIN {X 0,Y 422.949,Z 452.37,A -85,B 0,C 180,E1 -10007.154,E2 -10007.154} C_VEL
LIN {X 0,Y 424.139,Z 440.804,A -85,B 0,C 180,E1 -10008.225,E2 -10008.225} C_VEL
LIN {X 0,Y 425.065,Z 428.073,A -85,B 0,C 180,E1 -10009.184,E2 -10009.184} C_VEL
LIN {X 0,Y 425.969,Z 415.233,A -85,B 0,C 180,E1 -10009.932,E2 -10009.932} C_VEL
LIN {X 0,Y 426.612,Z 401.831,A -85,B 0,C 180,E1 -10010.523,E2 -10010.523} C_VEL
LIN {X 0,Y 427.117,Z 387.994,A -85,B 0,C 180,E1 -10010.938,E2 -10010.938} C_VEL
LIN {X 0,Y 427.694,Z 351.965,A -85,B 0,C 180,E1 -10011.54,E2 -10011.54} C_VEL
LIN {X 0,Y 428.636,Z 271.195,A -85,B 0,C 180,E1 -10012.835,E2 -10012.835} C_VEL
LIN {X 0,Y 423.23,Z 244.772,A -85,B 0,C 180,E1 -10013.64,E2 -10013.64} C_VEL
LIN {X 0,Y 423.197,Z 243.798,A -85,B 0,C 180,E1 -10013.745,E2 -10013.745} C_VEL
LIN {X 0,Y 424.609,Z 226.202,A -85,B 0,C 180,E1 -10016.782,E2 -10016.782} C_VEL
LIN {X 0,Y 421.461,Z 212.373,A -85,B 0,C 180,E1 -10019.555,E2 -10019.555} C_VEL
LIN {X 0,Y 418.253,Z 200.157,A -85,B 0,C 180,E1 -10022.17,E2 -10022.17} C_VEL
LIN {X 0,Y 418.258,Z 200.005,A -85,B 0,C 180,E1 -10024.84,E2 -10024.84} C_VEL
LIN {X 0,Y 418.255,Z 200.009,A -85,B 0,C 180,E1 -10028.44,E2 -10028.44} C_VEL
LIN {X 0,Y 418.237,Z 200.004,A -85,B 0,C 180,E1 -10032.232,E2 -10032.232} C_VEL
LIN {X 0,Y 418.234,Z 200.009,A -85,B 0,C 180,E1 -10035.108,E2 -10035.108} C_VEL
LIN {X 0,Y 418.236,Z 200.016,A -85,B 0,C 180,E1 -10037.766,E2 -10037.766} C_VEL
LIN {X 0,Y 418.247,Z 200.009,A -85,B 0,C 180,E1 -10041.557,E2 -10041.557} C_VEL
LIN {X 0,Y 418.255,Z 199.996,A -85,B 0,C 180,E1 -10045.158,E2 -10045.158} C_VEL
LIN {X 0,Y 418.241,Z 200.014,A -85,B 0,C 180,E1 -10047.471,E2 -10047.471} C_VEL
LIN {X 0,Y 418.271,Z 199.99,A -85,B 0,C 180,E1 -10050.893,E2 -10050.893} C_VEL
LIN {X 0,Y 418.265,Z 200.006,A -85,B 0,C 180,E1 -10054.095,E2 -10054.095} C_VEL
LIN {X 0,Y 418.232,Z 200.014,A -85,B 0,C 180,E1 -10057.263,E2 -10057.263} C_VEL
LIN {X 0,Y 418.277,Z 200.001,A -85,B 0,C 180,E1 -10060.364,E2 -10060.364} C_VEL
LIN {X 0,Y 418.31,Z 199.997,A -85,B 0,C 180,E1 -10063.404,E2 -10063.404} C_VEL
LIN {X 0,Y 418.34,Z 199.997,A -85,B 0,C 180,E1 -10066.999,E2 -10066.999} C_VEL
LIN {X 0,Y 418.334,Z 200.001,A -85,B 0,C 180,E1 -10070.328,E2 -10070.328} C_VEL
LIN {X 0,Y 418.506,Z 199.974,A -85,B 0,C 180,E1 -10072.279,E2 -10072.279} C_VEL
LIN {X 0,Y 418.506,Z 199.978,A -85,B 0,C 180,E1 -10074.217,E2 -10074.217} C_VEL
LIN {X 0,Y 418.537,Z 199.971,A -85,B 0,C 180,E1 -10078.075,E2 -10078.075} C_VEL
LIN {X 0,Y 418.665,Z 199.959,A -85,B 0,C 180,E1 -10080,E2 -10080} C_VEL
LIN {X 0,Y 418.504,Z 199.978,A -85,B 0,C 180,E1 -10082.888,E2 -10082.888} C_VEL
LIN {X 0,Y 418.486,Z 199.981,A -85,B 0,C 180,E1 -10086.751,E2 -10086.751} C_VEL
LIN {X 0,Y 418.393,Z 199.989,A -85,B 0,C 180,E1 -10088.695,E2 -10088.695} C_VEL
LIN {X 0,Y 418.308,Z 200.002,A -85,B 0,C 180,E1 -10091.631,E2 -10091.631} C_VEL
LIN {X 0,Y 418.295,Z 200.003,A -85,B 0,C 180,E1 -10094.597,E2 -10094.597} C_VEL
LIN {X 0,Y 418.281,Z 200.003,A -85,B 0,C 180,E1 -10097.604,E2 -10097.604} C_VEL
LIN {X 0,Y 418.243,Z 200.007,A -85,B 0,C 180,E1 -10100.663,E2 -10100.663} C_VEL
LIN {X 0,Y 418.281,Z 200.008,A -85,B 0,C 180,E1 -10103.781,E2 -10103.781} C_VEL
LIN {X 0,Y 418.303,Z 199.984,A -85,B 0,C 180,E1 -10107.071,E2 -10107.071} C_VEL
LIN {X 0,Y 418.238,Z 200.01,A -85,B 0,C 180,E1 -10110.272,E2 -10110.272} C_VEL
LIN {X 0,Y 418.242,Z 200.002,A -85,B 0,C 180,E1 -10113.678,E2 -10113.678} C_VEL
LIN {X 0,Y 418.234,Z 200.002,A -85,B 0,C 180,E1 -10117.225,E2 -10117.225} C_VEL
LIN {X 0,Y 418.249,Z 200.014,A -85,B 0,C 180,E1 -10119.682,E2 -10119.682} C_VEL
LIN {X 0,Y 418.223,Z 200.005,A -85,B 0,C 180,E1 -10122.322,E2 -10122.322} C_VEL
LIN {X 0,Y 418.23,Z 200.008,A -85,B 0,C 180,E1 -10125.109,E2 -10125.109} C_VEL
LIN {X 0,Y 418.235,Z 200.011,A -85,B 0,C 180,E1 -10127.767,E2 -10127.767} C_VEL
LIN {X 0,Y 418.237,Z 199.981,A -85,B 0,C 180,E1 -10130.622,E2 -10130.622} C_VEL
LIN {X 0,Y 418.238,Z 199.993,A -85,B 0,C 180,E1 -10133.976,E2 -10133.976} C_VEL
LIN {X 0,Y 418.266,Z 200.202,A -85,B 0,C 180,E1 -10136.054,E2 -10136.054} C_VEL
LIN {X 0,Y 422.389,Z 214.646,A -85,B 0,C 180,E1 -10138.75,E2 -10138.75} C_VEL
LIN {X 0,Y 425.713,Z 227.768,A -85,B 0,C 180,E1 -10141.041,E2 -10141.041} C_VEL
LIN {X 0,Y 426.166,Z 230.101,A -85,B 0,C 180,E1 -10141.43,E2 -10141.43} C_VEL
LIN {X 0,Y 424.857,Z 245.027,A -85,B 0,C 180,E1 -10143.572,E2 -10143.572} C_VEL
LIN {X 0,Y 429.24,Z 271.297,A -85,B 0,C 180,E1 -10144.361,E2 -10144.361} C_VEL
LIN {X 0,Y 426.84,Z 402.947,A -85,B 0,C 180,E1 -10146.725,E2 -10146.725} C_VEL
LIN {X 0,Y 426.247,Z 418.771,A -85,B 0,C 180,E1 -10147.14,E2 -10147.14} C_VEL
LIN {X 0,Y 425.42,Z 433.762,A -85,B 0,C 180,E1 -10147.726,E2 -10147.726} C_VEL
LIN {X 0,Y 424.421,Z 448.885,A -85,B 0,C 180,E1 -10148.528,E2 -10148.528} C_VEL
LIN {X 0,Y 423.32,Z 462.757,A -85,B 0,C 180,E1 -10149.469,E2 -10149.469} C_VEL
LIN {X 0,Y 422.187,Z 475.707,A -85,B 0,C 180,E1 -10150.554,E2 -10150.554} C_VEL
LIN {X 0,Y 421.097,Z 488.549,A -85,B 0,C 180,E1 -10151.863,E2 -10151.863} C_VEL
LIN {X 0,Y 420.157,Z 499.719,A -85,B 0,C 180,E1 -10153.23,E2 -10153.23} C_VEL
LIN {X 0,Y 419.204,Z 509.813,A -85,B 0,C 180,E1 -10154.69,E2 -10154.69} C_VEL
LIN {X 0,Y 418.418,Z 519.686,A -85,B 0,C 180,E1 -10156.4,E2 -10156.4} C_VEL
LIN {X 0,Y 417.863,Z 527.9,A -85,B 0,C 180,E1 -10158.111,E2 -10158.111} C_VEL
LIN {X 0,Y 417.457,Z 534.708,A -85,B 0,C 180,E1 -10159.819,E2 -10159.819} C_VEL
LIN {X 0,Y 417.211,Z 540.944,A -85,B 0,C 180,E1 -10161.768,E2 -10161.768} C_VEL
LIN {X 0,Y 417.114,Z 545.847,A -85,B 0,C 180,E1 -10163.77,E2 -10163.77} C_VEL
LIN {X 0,Y 417.061,Z 548.388,A -85,B 0,C 180,E1 -10165.167,E2 -10165.167} C_VEL
LIN {X 0,Y 417.086,Z 550.868,A -85,B 0,C 180,E1 -10167.103,E2 -10167.103} C_VEL
LIN {X 0,Y 417.053,Z 552.11,A -85,B 0,C 180,E1 -10169.035,E2 -10169.035} C_VEL
LIN {X 0,Y 417.053,Z 552.108,A -85,B 0,C 180,E1 -10170.966,E2 -10170.966} C_VEL
LIN {X 0,Y 417.087,Z 550.86,A -85,B 0,C 180,E1 -10172.898,E2 -10172.898} C_VEL
LIN {X 0,Y 417.091,Z 548.378,A -85,B 0,C 180,E1 -10174.833,E2 -10174.833} C_VEL
LIN {X 0,Y 417.163,Z 544.617,A -85,B 0,C 180,E1 -10176.773,E2 -10176.773} C_VEL
LIN {X 0,Y 417.259,Z 539.481,A -85,B 0,C 180,E1 -10178.719,E2 -10178.719} C_VEL
LIN {X 0,Y 417.597,Z 532.847,A -85,B 0,C 180,E1 -10180.669,E2 -10180.669} C_VEL
LIN {X 0,Y 418.122,Z 524.529,A -85,B 0,C 180,E1 -10182.622,E2 -10182.622} C_VEL
LIN {X 0,Y 418.754,Z 515.642,A -85,B 0,C 180,E1 -10184.333,E2 -10184.333} C_VEL
LIN {X 0,Y 419.621,Z 504.932,A -85,B 0,C 180,E1 -10186.043,E2 -10186.043} C_VEL
LIN {X 0,Y 420.576,Z 493.93,A -85,B 0,C 180,E1 -10187.505,E2 -10187.505} C_VEL
LIN {X 0,Y 421.601,Z 481.905,A -85,B 0,C 180,E1 -10188.843,E2 -10188.843} C_VEL
LIN {X 0,Y 422.776,Z 468.744,A -85,B 0,C 180,E1 -10190.051,E2 -10190.051} C_VEL
LIN {X 0,Y 423.839,Z 455.962,A -85,B 0,C 180,E1 -10191.013,E2 -10191.013} C_VEL
LIN {X 0,Y 424.913,Z 441.56,A -85,B 0,C 180,E1 -10191.882,E2 -10191.882} C_VEL
LIN {X 0,Y 425.797,Z 426.799,A -85,B 0,C 180,E1 -10192.566,E2 -10192.566} C_VEL
LIN {X 0,Y 426.52,Z 411.548,A -85,B 0,C 180,E1 -10193.07,E2 -10193.07} C_VEL
LIN {X 0,Y 427.098,Z 391.167,A -85,B 0,C 180,E1 -10193.486,E2 -10193.486} C_VEL
LIN {X 0,Y 429.215,Z 271.326,A -85,B 0,C 180,E1 -10195.632,E2 -10195.632} C_VEL
LIN {X 0,Y 424.854,Z 244.981,A -85,B 0,C 180,E1 -10196.424,E2 -10196.424} C_VEL
LIN {X 0,Y 426.208,Z 230.112,A -85,B 0,C 180,E1 -10198.568,E2 -10198.568} C_VEL
LIN {X 0,Y 423.1,Z 217.163,A -85,B 0,C 180,E1 -10200.794,E2 -10200.794} C_VEL
